C08945=1021.855,337.946,-141.506,171.172,49.202,159.657
C08946=1021.848,337.709,-141.471,171.166,49.204,159.656
C08947=1021.841,337.470,-141.437,171.159,49.205,159.655
C08948=1021.835,337.231,-141.402,171.152,49.207,159.655
C08949=1021.827,336.993,-141.367,171.146,49.209,159.654
C08950=1021.820,336.754,-141.333,171.140,49.210,159.654
C08951=1021.813,336.516,-141.298,171.134,49.211,159.653
C08952=1021.806,336.277,-141.264,171.128,49.213,159.652
C08953=1021.799,336.030,-141.228,171.121,49.214,159.652
C08954=1021.791,335.783,-141.192,171.115,49.216,159.651
C08955=1021.784,335.536,-141.157,171.108,49.218,159.651
C08956=1021.777,335.288,-141.121,171.101,49.219,159.650
C08957=1021.770,335.041,-141.086,171.095,49.221,159.649
C08958=1021.762,334.793,-141.049,171.089,49.223,159.649
C08959=1021.755,334.546,-141.014,171.082,49.225,159.648
C08960=1021.748,334.299,-140.978,171.076,49.226,159.647
C08961=1021.741,334.051,-140.943,171.070,49.228,159.647
C08962=1021.734,333.804,-140.907,171.063,49.229,159.646
C08963=1021.727,333.556,-140.871,171.057,49.231,159.646
C08964=1021.719,333.310,-140.836,171.050,49.233,159.645
C08965=1021.713,333.062,-140.800,171.044,49.235,159.645
C08966=1021.705,332.814,-140.765,171.038,49.237,159.644
C08967=1021.699,332.567,-140.730,171.031,49.238,159.643
C08968=1021.691,332.320,-140.694,171.024,49.240,159.643
C08969=1021.683,332.072,-140.659,171.018,49.242,159.642
C08970=1021.677,331.825,-140.624,171.012,49.244,159.642
C08971=1021.670,331.578,-140.589,171.006,49.246,159.641
C08972=1021.662,331.330,-140.553,171.000,49.248,159.641
C08973=1021.655,331.082,-140.519,170.993,49.250,159.640
C08974=1021.648,330.836,-140.483,170.987,49.252,159.640
C08975=1021.641,330.588,-140.448,170.980,49.253,159.639
C08976=1021.634,330.340,-140.412,170.974,49.255,159.639
C08977=1021.626,330.093,-140.378,170.968,49.257,159.638
C08978=1021.619,329.846,-140.343,170.961,49.259,159.638
C08979=1021.613,329.599,-140.307,170.955,49.261,159.637
C08980=1021.605,329.350,-140.272,170.949,49.263,159.637
C08981=1021.598,329.103,-140.237,170.943,49.265,159.636
C08982=1021.591,328.856,-140.202,170.937,49.267,159.636
C08983=1021.584,328.609,-140.167,170.930,49.269,159.635
C08984=1021.578,328.361,-140.132,170.924,49.271,159.635
C08985=1021.570,328.113,-140.098,170.918,49.272,159.634
C08986=1021.563,327.866,-140.063,170.912,49.274,159.634
C08987=1021.556,327.618,-140.028,170.906,49.276,159.633
C08988=1021.549,327.371,-139.992,170.900,49.278,159.633
C08989=1021.542,327.124,-139.958,170.894,49.280,159.632
C08990=1021.535,326.876,-139.923,170.887,49.283,159.632
C08991=1021.529,326.628,-139.888,170.881,49.285,159.631
C08992=1021.521,326.381,-139.854,170.875,49.287,159.631
C08993=1021.514,326.134,-139.819,170.869,49.289,159.630
C08994=1021.506,325.886,-139.785,170.863,49.291,159.630
C08995=1021.499,325.639,-139.750,170.856,49.294,159.630
C08996=1021.492,325.391,-139.716,170.850,49.296,159.629
C08997=1021.484,325.144,-139.682,170.844,49.298,159.629
C08998=1021.478,324.896,-139.647,170.838,49.300,159.628
C08999=1021.470,324.649,-139.613,170.832,49.302,159.628
C09000=1021.463,324.401,-139.579,170.826,49.304,159.627
C09001=1021.457,324.153,-139.544,170.819,49.306,159.627
C09002=1021.449,323.906,-139.510,170.814,49.309,159.626
C09003=1021.442,323.658,-139.476,170.808,49.311,159.626
C09004=1021.435,323.411,-139.441,170.802,49.314,159.626
C09005=1021.428,323.170,-139.408,170.796,49.315,159.625
C09006=1021.421,322.930,-139.375,170.790,49.317,159.625
C09007=1021.414,322.689,-139.342,170.784,49.320,159.624
C09008=1021.408,322.449,-139.309,170.778,49.322,159.624
C09009=1021.401,322.208,-139.275,170.773,49.325,159.624
C09010=1021.394,321.967,-139.242,170.767,49.326,159.623
C09011=1021.387,321.727,-139.209,170.761,49.329,159.623
C09012=1021.380,321.486,-139.175,170.755,49.331,159.622
C09013=1021.373,321.239,-139.142,170.749,49.334,159.622
C09014=1021.366,320.991,-139.108,170.743,49.336,159.622
C09015=1021.360,320.743,-139.073,170.737,49.338,159.621
C09016=1021.352,320.496,-139.039,170.731,49.340,159.621
C09017=1021.345,320.248,-139.005,170.726,49.343,159.621
C09018=1021.338,320.000,-138.971,170.720,49.345,159.620
C09019=1021.331,319.753,-138.937,170.713,49.347,159.620
C09020=1021.325,319.506,-138.903,170.707,49.350,159.620
C09021=1021.317,319.258,-138.870,170.701,49.352,159.619
C09022=1021.311,319.010,-138.835,170.696,49.355,159.619
C09023=1021.304,318.762,-138.801,170.690,49.357,159.619
C09024=1021.297,318.515,-138.768,170.684,49.359,159.618
C09025=1021.291,318.267,-138.733,170.678,49.362,159.618
C09026=1021.284,318.020,-138.700,170.673,49.364,159.617
C09027=1021.276,317.772,-138.666,170.667,49.367,159.617
C09028=1021.270,317.525,-138.632,170.661,49.369,159.617
C09029=1021.263,317.277,-138.598,170.655,49.371,159.616
C09030=1021.256,317.029,-138.564,170.650,49.374,159.616
C09031=1021.249,316.782,-138.530,170.644,49.377,159.616
C09032=1021.242,316.535,-138.497,170.638,49.379,159.615
C09033=1021.236,316.287,-138.462,170.632,49.381,159.615
C09034=1021.229,316.039,-138.429,170.627,49.384,159.615
C09035=1021.222,315.792,-138.396,170.620,49.387,159.614
C09036=1021.215,315.544,-138.362,170.614,49.389,159.614
C09037=1021.209,315.297,-138.328,170.609,49.392,159.614
C09038=1021.202,315.049,-138.294,170.603,49.394,159.614
C09039=1021.195,314.801,-138.260,170.597,49.396,159.613
C09040=1021.189,314.553,-138.227,170.591,49.399,159.613
C09041=1021.182,314.306,-138.193,170.585,49.401,159.613
C09042=1021.175,314.059,-138.160,170.580,49.404,159.612
C09043=1021.168,313.811,-138.126,170.574,49.407,159.612
C09044=1021.163,313.563,-138.093,170.568,49.409,159.612
C09045=1021.156,313.315,-138.059,170.563,49.412,159.611
C09046=1021.149,313.069,-138.025,170.557,49.414,159.611
C09047=1021.142,312.820,-137.992,170.551,49.417,159.611
C09048=1021.136,312.573,-137.958,170.546,49.420,159.611
C09049=1021.129,312.325,-137.924,170.540,49.422,159.610
C09050=1021.123,312.078,-137.892,170.534,49.425,159.610
C09051=1021.115,311.830,-137.858,170.529,49.427,159.610
C09052=1021.109,311.582,-137.825,170.523,49.430,159.609
C09053=1021.103,311.334,-137.791,170.517,49.433,159.609
C09054=1021.096,311.087,-137.758,170.512,49.435,159.609
C09055=1021.090,310.840,-137.724,170.506,49.438,159.609
C09056=1021.083,310.592,-137.691,170.502,49.441,159.608
C09057=1021.077,310.344,-137.657,170.496,49.443,159.608
C09058=1021.070,310.096,-137.624,170.490,49.446,159.608
C09059=1021.064,309.849,-137.591,170.485,49.448,159.608
C09060=1021.057,309.602,-137.558,170.478,49.452,159.607
C09061=1021.050,309.353,-137.525,170.473,49.455,159.607
C09062=1021.043,309.106,-137.493,170.467,49.458,159.607
C09063=1021.036,308.858,-137.460,170.462,49.460,159.607
C09064=1021.029,308.610,-137.427,170.456,49.463,159.606
C09065=1021.023,308.372,-137.396,170.451,49.466,159.606
C09066=1021.016,308.134,-137.364,170.446,49.468,159.606
C09067=1021.009,307.896,-137.333,170.441,49.472,159.606
C09068=1021.003,307.658,-137.301,170.435,49.474,159.606
C09069=1020.996,307.420,-137.270,170.429,49.477,159.606
C09070=1020.990,307.182,-137.238,170.424,49.480,159.605
C09071=1020.984,306.944,-137.207,170.419,49.482,159.605
C09072=1020.977,306.706,-137.176,170.414,49.486,159.605
C09073=1020.970,306.459,-137.144,170.409,49.488,159.605
C09074=1020.963,306.210,-137.111,170.403,49.491,159.605
C09075=1020.956,305.963,-137.079,170.398,49.495,159.605
C09076=1020.950,305.715,-137.046,170.392,49.497,159.604
C09077=1020.943,305.467,-137.013,170.387,49.501,159.604
C09078=1020.936,305.220,-136.981,170.381,49.503,159.604
C09079=1020.930,304.972,-136.948,170.376,49.506,159.604
C09080=1020.922,304.724,-136.916,170.371,49.510,159.604
C09081=1020.916,304.476,-136.883,170.365,49.512,159.603
C09082=1020.910,304.229,-136.851,170.360,49.515,159.603
C09083=1020.903,303.981,-136.818,170.354,49.519,159.603
C09084=1020.896,303.734,-136.786,170.349,49.521,159.603
C09085=1020.889,303.485,-136.754,170.343,49.525,159.603
C09086=1020.883,303.237,-136.721,170.338,49.528,159.603
C09087=1020.876,302.990,-136.688,170.333,49.531,159.603
C09088=1020.869,302.743,-136.656,170.327,49.534,159.602
C09089=1020.863,302.494,-136.624,170.322,49.537,159.602
C09090=1020.856,302.246,-136.592,170.316,49.540,159.602
C09091=1020.849,301.999,-136.559,170.311,49.543,159.602
C09092=1020.843,301.751,-136.527,170.306,49.547,159.602
C09093=1020.836,301.503,-136.495,170.300,49.549,159.602
C09094=1020.830,301.256,-136.462,170.295,49.552,159.602
C09095=1020.823,301.008,-136.431,170.290,49.556,159.602
C09096=1020.817,300.760,-136.398,170.284,49.559,159.601
C09097=1020.810,300.512,-136.365,170.279,49.562,159.601
C09098=1020.803,300.264,-136.333,170.274,49.565,159.601
C09099=1020.797,300.016,-136.301,170.268,49.568,159.601
C09100=1020.790,299.768,-136.269,170.263,49.571,159.601
C09101=1020.784,299.521,-136.236,170.257,49.575,159.601
C09102=1020.778,299.273,-136.204,170.252,49.578,159.601
C09103=1020.771,299.025,-136.172,170.247,49.581,159.601
C09104=1020.765,298.777,-136.140,170.241,49.584,159.600
C09105=1020.758,298.530,-136.108,170.236,49.588,159.600
C09106=1020.752,298.282,-136.076,170.231,49.591,159.600
C09107=1020.745,298.034,-136.044,170.225,49.594,159.600
C09108=1020.739,297.786,-136.012,170.220,49.597,159.600
C09109=1020.733,297.538,-135.980,170.215,49.601,159.600
C09110=1020.726,297.291,-135.948,170.211,49.603,159.600
C09111=1020.720,297.042,-135.916,170.205,49.607,159.600
C09112=1020.713,296.795,-135.884,170.200,49.610,159.600
C09113=1020.707,296.547,-135.851,170.195,49.613,159.600
C09114=1020.700,296.299,-135.820,170.189,49.617,159.600
C09115=1020.694,296.051,-135.788,170.184,49.620,159.599
C09116=1020.689,295.804,-135.756,170.179,49.623,159.599
C09117=1020.682,295.556,-135.724,170.174,49.627,159.599
C09118=1020.676,295.308,-135.692,170.168,49.630,159.599
C09119=1020.669,295.061,-135.660,170.163,49.633,159.599
C09120=1020.663,294.812,-135.628,170.158,49.637,159.599
C09121=1020.657,294.564,-135.596,170.153,49.640,159.599
C09122=1020.650,294.316,-135.565,170.148,49.643,159.599
C09123=1020.644,294.068,-135.533,170.143,49.647,159.599
C09124=1020.638,293.821,-135.501,170.138,49.650,159.599
C09125=1020.632,293.592,-135.471,170.133,49.653,159.599
C09126=1020.627,293.362,-135.442,170.128,49.656,159.599
C09127=1020.620,293.133,-135.413,170.123,49.659,159.599
C09128=1020.614,292.904,-135.384,170.119,49.662,159.599
C09129=1020.608,292.674,-135.355,170.113,49.666,159.599
C09130=1020.603,292.445,-135.325,170.110,49.669,159.599
C09131=1020.596,292.216,-135.296,170.104,49.673,159.599
C09132=1020.590,291.986,-135.268,170.100,49.675,159.599
C09133=1020.584,291.738,-135.236,170.095,49.679,159.599
C09134=1020.578,291.490,-135.204,170.090,49.683,159.599
C09135=1020.571,291.242,-135.173,170.084,49.686,159.599
C09136=1020.565,290.995,-135.142,170.079,49.690,159.599
C09137=1020.558,290.747,-135.110,170.074,49.693,159.599
C09138=1020.552,290.499,-135.079,170.069,49.697,159.599
C09139=1020.545,290.251,-135.048,170.064,49.700,159.599
C09140=1020.539,290.004,-135.017,170.059,49.704,159.599
C09141=1020.533,289.756,-134.985,170.054,49.707,159.599
C09142=1020.526,289.507,-134.954,170.049,49.711,159.599
C09143=1020.520,289.259,-134.923,170.044,49.715,159.599
C09144=1020.514,289.012,-134.892,170.038,49.719,159.599
C09145=1020.507,288.763,-134.861,170.034,49.722,159.599
C09146=1020.500,288.515,-134.830,170.028,49.726,159.599
C09147=1020.494,288.268,-134.798,170.023,49.730,159.599
C09148=1020.488,288.020,-134.768,170.018,49.734,159.599
C09149=1020.481,287.772,-134.736,170.014,49.736,159.599
C09150=1020.474,287.524,-134.705,170.009,49.740,159.599
C09151=1020.469,287.276,-134.675,170.004,49.744,159.599
C09152=1020.462,287.028,-134.643,169.999,49.748,159.599
C09153=1020.455,286.780,-134.612,169.994,49.752,159.599
C09154=1020.449,286.533,-134.581,169.989,49.755,159.599
C09155=1020.443,286.284,-134.551,169.984,49.759,159.599
C09156=1020.436,286.036,-134.519,169.979,49.763,159.599
C09157=1020.430,285.788,-134.489,169.974,49.767,159.599
C09158=1020.424,285.540,-134.457,169.969,49.771,159.599
C09159=1020.417,285.292,-134.427,169.964,49.774,159.599
C09160=1020.411,285.045,-134.396,169.959,49.778,159.599
C09161=1020.405,284.796,-134.365,169.954,49.782,159.600
C09162=1020.399,284.548,-134.335,169.949,49.786,159.599
C09163=1020.392,284.300,-134.303,169.944,49.789,159.600
C09164=1020.386,284.052,-134.272,169.939,49.793,159.600
C09165=1020.379,283.804,-134.243,169.934,49.797,159.600
C09166=1020.373,283.556,-134.212,169.929,49.801,159.600
C09167=1020.367,283.309,-134.181,169.924,49.805,159.600
C09168=1020.360,283.060,-134.150,169.919,49.809,159.600
C09169=1020.354,282.812,-134.119,169.914,49.813,159.600
C09170=1020.347,282.564,-134.090,169.909,49.817,159.600
C09171=1020.341,282.316,-134.058,169.904,49.821,159.600
C09172=1020.335,282.068,-134.028,169.899,49.825,159.600
C09173=1020.328,281.820,-133.997,169.895,49.829,159.600
C09174=1020.322,281.572,-133.967,169.890,49.833,159.600
C09175=1020.315,281.324,-133.937,169.886,49.836,159.601
C09176=1020.309,281.076,-133.906,169.881,49.840,159.601
C09177=1020.303,280.827,-133.876,169.876,49.845,159.601
C09178=1020.297,280.580,-133.845,169.871,49.849,159.601
C09179=1020.290,280.332,-133.814,169.866,49.853,159.601
C09180=1020.284,280.084,-133.784,169.861,49.857,159.601
C09181=1020.278,279.836,-133.753,169.856,49.861,159.601
C09182=1020.272,279.588,-133.723,169.852,49.865,159.601
C09183=1020.265,279.340,-133.693,169.847,49.868,159.602
C09184=1020.259,279.092,-133.663,169.842,49.872,159.602
C09185=1020.254,278.869,-133.635,169.838,49.876,159.602
C09186=1020.247,278.645,-133.608,169.833,49.880,159.602
C09187=1020.242,278.422,-133.581,169.829,49.884,159.602
C09188=1020.237,278.199,-133.553,169.825,49.887,159.602
C09189=1020.231,277.976,-133.526,169.820,49.891,159.602
C09190=1020.226,277.753,-133.499,169.816,49.895,159.603
C09191=1020.219,277.529,-133.472,169.812,49.898,159.603
C09192=1020.214,277.306,-133.444,169.807,49.902,159.603
C09193=1020.209,277.058,-133.414,169.802,49.906,159.603
C09194=1020.201,276.810,-133.384,169.797,49.910,159.603
C09195=1020.196,276.562,-133.353,169.792,49.914,159.603
C09196=1020.189,276.314,-133.324,169.788,49.919,159.603
C09197=1020.183,276.066,-133.293,169.783,49.923,159.603
C09198=1020.176,275.818,-133.264,169.778,49.927,159.604
C09199=1020.171,275.570,-133.234,169.774,49.931,159.604
C09200=1020.163,275.322,-133.203,169.769,49.935,159.604
C09201=1020.158,275.073,-133.174,169.764,49.940,159.604
C09202=1020.152,274.825,-133.143,169.759,49.944,159.604
C09203=1020.145,274.577,-133.113,169.755,49.948,159.604
C09204=1020.139,274.329,-133.084,169.751,49.952,159.605
C09205=1020.133,274.081,-133.054,169.746,49.957,159.605
C09206=1020.126,273.833,-133.023,169.741,49.961,159.605
C09207=1020.120,273.584,-132.994,169.737,49.965,159.605
C09208=1020.114,273.337,-132.964,169.732,49.969,159.605
C09209=1020.107,273.088,-132.934,169.727,49.974,159.606
C09210=1020.102,272.840,-132.904,169.722,49.978,159.606
C09211=1020.095,272.592,-132.874,169.718,49.982,159.606
C09212=1020.090,272.344,-132.845,169.713,49.986,159.606
C09213=1020.082,272.096,-132.815,169.708,49.991,159.606
C09214=1020.076,271.848,-132.786,169.704,49.995,159.607
C09215=1020.070,271.600,-132.755,169.699,49.999,159.607
C09216=1020.064,271.352,-132.726,169.694,50.004,159.607
C09217=1020.058,271.103,-132.696,169.690,50.009,159.607
C09218=1020.051,270.855,-132.666,169.685,50.013,159.607
C09219=1020.046,270.607,-132.637,169.680,50.017,159.608
C09220=1020.039,270.359,-132.607,169.676,50.022,159.608
C09221=1020.033,270.111,-132.578,169.671,50.026,159.608
C09222=1020.027,269.862,-132.547,169.666,50.030,159.608
C09223=1020.020,269.614,-132.518,169.662,50.035,159.609
C09224=1020.015,269.366,-132.489,169.657,50.039,159.609
C09225=1020.009,269.118,-132.460,169.652,50.044,159.609
C09226=1020.002,268.870,-132.430,169.648,50.048,159.609
C09227=1019.996,268.622,-132.401,169.643,50.053,159.610
C09228=1019.990,268.373,-132.371,169.638,50.057,159.610
C09229=1019.984,268.125,-132.342,169.634,50.061,159.610
C09230=1019.977,267.877,-132.312,169.629,50.066,159.610
C09231=1019.971,267.629,-132.282,169.624,50.071,159.610
C09232=1019.965,267.381,-132.253,169.620,50.075,159.611
C09233=1019.959,267.133,-132.224,169.615,50.080,159.611
C09234=1019.953,266.885,-132.195,169.611,50.085,159.611
C09235=1019.946,266.636,-132.164,169.606,50.089,159.612
C09236=1019.940,266.388,-132.135,169.602,50.094,159.612
C09237=1019.934,266.140,-132.106,169.597,50.098,159.612
C09238=1019.928,265.892,-132.077,169.593,50.103,159.612
C09239=1019.921,265.643,-132.048,169.588,50.107,159.612
C09240=1019.916,265.395,-132.019,169.583,50.112,159.613
C09241=1019.910,265.147,-131.990,169.579,50.116,159.613
C09242=1019.903,264.899,-131.961,169.574,50.121,159.613
C09243=1019.897,264.651,-131.932,169.570,50.126,159.614
C09244=1019.891,264.402,-131.903,169.565,50.131,159.614
C09245=1019.885,264.182,-131.876,169.560,50.135,159.614
C09246=1019.880,263.961,-131.851,169.557,50.139,159.615
C09247=1019.874,263.740,-131.825,169.553,50.143,159.615
C09248=1019.868,263.519,-131.799,169.548,50.147,159.615
C09249=1019.863,263.298,-131.773,169.545,50.152,159.615
C09250=1019.857,263.078,-131.747,169.541,50.155,159.615
C09251=1019.852,262.856,-131.722,169.537,50.160,159.616
C09252=1019.846,262.636,-131.696,169.533,50.164,159.616
C09253=1019.841,262.387,-131.666,169.528,50.169,159.616
C09254=1019.835,262.139,-131.637,169.524,50.174,159.617
C09255=1019.829,261.890,-131.609,169.519,50.178,159.617
C09256=1019.822,261.642,-131.580,169.515,50.183,159.617
C09257=1019.816,261.394,-131.551,169.511,50.188,159.618
C09258=1019.810,261.146,-131.522,169.506,50.193,159.618
C09259=1019.804,260.898,-131.493,169.502,50.198,159.618
C09260=1019.798,260.649,-131.464,169.497,50.202,159.619
C09261=1019.791,260.401,-131.435,169.493,50.207,159.619
C09262=1019.785,260.153,-131.406,169.488,50.212,159.619
C09263=1019.779,259.905,-131.377,169.484,50.217,159.620
C09264=1019.773,259.656,-131.349,169.478,50.222,159.620
C09265=1019.766,259.408,-131.320,169.474,50.227,159.620
C09266=1019.760,259.159,-131.292,169.470,50.232,159.620
C09267=1019.754,258.912,-131.263,169.465,50.237,159.621
C09268=1019.748,258.664,-131.236,169.461,50.242,159.621
C09269=1019.741,258.415,-131.207,169.457,50.247,159.622
C09270=1019.736,258.167,-131.178,169.452,50.252,159.622
C09271=1019.729,257.919,-131.150,169.448,50.257,159.622
C09272=1019.723,257.670,-131.121,169.444,50.262,159.623
C09273=1019.716,257.422,-131.092,169.438,50.267,159.623
C09274=1019.710,257.173,-131.065,169.434,50.272,159.623
C09275=1019.703,256.925,-131.036,169.430,50.277,159.624
C09276=1019.697,256.677,-131.007,169.425,50.282,159.624
C09277=1019.690,256.429,-130.979,169.421,50.287,159.625
C09278=1019.685,256.180,-130.951,169.417,50.293,159.625
C09279=1019.679,255.932,-130.923,169.412,50.297,159.625
C09280=1019.672,255.684,-130.894,169.408,50.303,159.626
C09281=1019.666,255.435,-130.866,169.403,50.308,159.626
C09282=1019.660,255.187,-130.838,169.399,50.313,159.627
C09283=1019.653,254.939,-130.809,169.394,50.318,159.627
C09284=1019.647,254.690,-130.781,169.390,50.323,159.627
C09285=1019.642,254.442,-130.753,169.386,50.328,159.628
C09286=1019.635,254.194,-130.724,169.381,50.333,159.628
C09287=1019.629,253.945,-130.696,169.377,50.338,159.628
C09288=1019.623,253.697,-130.668,169.373,50.343,159.629
C09289=1019.616,253.448,-130.640,169.368,50.348,159.629
C09290=1019.611,253.201,-130.611,169.363,50.354,159.630
C09291=1019.605,252.952,-130.583,169.359,50.359,159.630
C09292=1019.598,252.704,-130.555,169.355,50.364,159.631
C09293=1019.592,252.455,-130.527,169.350,50.369,159.631
C09294=1019.586,252.207,-130.498,169.346,50.374,159.631
C09295=1019.580,251.959,-130.470,169.342,50.380,159.632
C09296=1019.574,251.710,-130.442,169.338,50.385,159.632
C09297=1019.568,251.461,-130.414,169.333,50.390,159.633
C09298=1019.562,251.214,-130.386,169.329,50.395,159.633
C09299=1019.556,250.966,-130.357,169.324,50.401,159.633
C09300=1019.550,250.717,-130.329,169.320,50.406,159.634
C09301=1019.543,250.468,-130.301,169.316,50.411,159.634
C09302=1019.538,250.220,-130.273,169.311,50.416,159.635
C09303=1019.532,249.972,-130.245,169.307,50.422,159.635
C09304=1019.525,249.723,-130.217,169.303,50.427,159.636
C09305=1019.520,249.502,-130.192,169.299,50.432,159.636
C09306=1019.515,249.280,-130.167,169.295,50.437,159.636
C09307=1019.510,249.058,-130.143,169.292,50.441,159.637
C09308=1019.504,248.837,-130.117,169.287,50.446,159.637
C09309=1019.499,248.614,-130.092,169.284,50.451,159.638
C09310=1019.493,248.393,-130.067,169.280,50.455,159.638
C09311=1019.488,248.171,-130.042,169.276,50.460,159.638
C09312=1019.483,247.950,-130.017,169.272,50.465,159.639
C09313=1019.476,247.702,-129.989,169.268,50.470,159.639
C09314=1019.471,247.454,-129.961,169.264,50.476,159.640
C09315=1019.464,247.205,-129.933,169.260,50.481,159.640
C09316=1019.458,246.956,-129.906,169.256,50.486,159.641
C09317=1019.453,246.708,-129.878,169.251,50.491,159.641
C09318=1019.446,246.459,-129.850,169.247,50.496,159.641
C09319=1019.441,246.211,-129.822,169.242,50.502,159.642
C09320=1019.435,245.962,-129.794,169.238,50.508,159.642
C09321=1019.429,245.714,-129.766,169.234,50.513,159.643
C09322=1019.423,245.466,-129.738,169.229,50.518,159.643
C09323=1019.417,245.217,-129.710,169.225,50.524,159.643
C09324=1019.411,244.969,-129.682,169.221,50.529,159.644
C09325=1019.405,244.721,-129.654,169.217,50.534,159.644
C09326=1019.399,244.473,-129.627,169.213,50.540,159.645
C09327=1019.393,244.224,-129.599,169.209,50.546,159.646
C09328=1019.388,243.976,-129.571,169.204,50.551,159.646
C09329=1019.381,243.727,-129.543,169.200,50.557,159.646
C09330=1019.376,243.479,-129.515,169.196,50.562,159.647
C09331=1019.370,243.230,-129.487,169.192,50.567,159.647
C09332=1019.364,242.982,-129.460,169.188,50.573,159.648
C09333=1019.358,242.733,-129.433,169.184,50.578,159.648
C09334=1019.352,242.485,-129.405,169.180,50.584,159.649
C09335=1019.346,242.236,-129.378,169.175,50.590,159.649
C09336=1019.340,241.989,-129.350,169.171,50.595,159.650
C09337=1019.334,241.740,-129.322,169.166,50.601,159.650
C09338=1019.328,241.492,-129.295,169.163,50.607,159.651
C09339=1019.322,241.243,-129.268,169.159,50.612,159.651
C09340=1019.316,240.994,-129.240,169.153,50.618,159.652
C09341=1019.310,240.746,-129.213,169.150,50.624,159.652
C09342=1019.304,240.498,-129.185,169.146,50.629,159.653
C09343=1019.298,240.249,-129.158,169.141,50.635,159.653
C09344=1019.292,240.001,-129.130,169.138,50.641,159.654
C09345=1019.286,239.753,-129.104,169.133,50.646,159.654
C09346=1019.280,239.504,-129.075,169.129,50.652,159.655
C09347=1019.275,239.256,-129.049,169.125,50.658,159.656
C09348=1019.268,239.007,-129.021,169.121,50.663,159.656
C09349=1019.262,238.759,-128.994,169.117,50.669,159.657
C09350=1019.256,238.510,-128.966,169.112,50.675,159.657
C09351=1019.250,238.262,-128.939,169.108,50.681,159.658
C09352=1019.245,238.013,-128.913,169.104,50.686,159.658
C09353=1019.238,237.765,-128.885,169.100,50.692,159.659
C09354=1019.232,237.517,-128.858,169.095,50.698,159.659
C09355=1019.226,237.268,-128.831,169.091,50.704,159.660
C09356=1019.220,237.020,-128.804,169.087,50.710,159.660
C09357=1019.214,236.771,-128.777,169.083,50.716,159.661
C09358=1019.208,236.522,-128.750,169.079,50.722,159.662
C09359=1019.202,236.274,-128.724,169.075,50.727,159.662
C09360=1019.195,236.026,-128.696,169.071,50.734,159.663
C09361=1019.189,235.777,-128.669,169.066,50.739,159.663
C09362=1019.184,235.529,-128.643,169.062,50.745,159.664
C09363=1019.177,235.280,-128.616,169.059,50.751,159.664
C09364=1019.171,235.032,-128.588,169.054,50.757,159.665
C09365=1019.166,234.807,-128.564,169.051,50.763,159.666
C09366=1019.160,234.581,-128.540,169.047,50.768,159.666
C09367=1019.155,234.356,-128.515,169.043,50.774,159.667
C09368=1019.150,234.132,-128.491,169.039,50.779,159.667
C09369=1019.145,233.907,-128.467,169.035,50.784,159.668
C09370=1019.139,233.682,-128.442,169.031,50.790,159.668
C09371=1019.134,233.457,-128.418,169.029,50.795,159.669
C09372=1019.128,233.232,-128.394,169.024,50.801,159.669
C09373=1019.122,232.983,-128.367,169.021,50.807,159.670
C09374=1019.116,232.735,-128.340,169.016,50.812,159.670
C09375=1019.110,232.487,-128.314,169.012,50.819,159.671
C09376=1019.104,232.238,-128.287,169.008,50.825,159.672
C09377=1019.098,231.989,-128.260,169.004,50.831,159.672
C09378=1019.092,231.741,-128.233,169.000,50.837,159.673
C09379=1019.086,231.493,-128.206,168.996,50.843,159.673
C09380=1019.080,231.245,-128.179,168.992,50.849,159.674
C09381=1019.074,230.996,-128.152,168.987,50.855,159.675
C09382=1019.068,230.747,-128.126,168.984,50.861,159.675
C09383=1019.062,230.499,-128.099,168.980,50.867,159.676
C09384=1019.057,230.251,-128.072,168.975,50.874,159.676
C09385=1019.050,230.001,-128.045,168.972,50.880,159.677
C09386=1019.044,229.753,-128.019,168.968,50.886,159.678
C09387=1019.039,229.504,-127.993,168.963,50.892,159.678
C09388=1019.033,229.256,-127.966,168.959,50.898,159.679
C09389=1019.027,229.007,-127.939,168.955,50.904,159.680
C09390=1019.020,228.759,-127.913,168.951,50.910,159.680
C09391=1019.015,228.510,-127.886,168.947,50.916,159.681
C09392=1019.009,228.262,-127.860,168.943,50.922,159.681
C09393=1019.003,228.014,-127.833,168.939,50.929,159.682
C09394=1018.997,227.765,-127.806,168.935,50.935,159.683
C09395=1018.992,227.516,-127.780,168.932,50.942,159.684
C09396=1018.985,227.268,-127.754,168.927,50.948,159.684
C09397=1018.979,227.019,-127.727,168.923,50.954,159.685
C09398=1018.973,226.771,-127.701,168.919,50.961,159.685
C09399=1018.968,226.522,-127.675,168.915,50.967,159.686
C09400=1018.961,226.274,-127.649,168.911,50.973,159.687
C09401=1018.955,226.025,-127.622,168.906,50.979,159.687
C09402=1018.950,225.777,-127.595,168.903,50.985,159.688
C09403=1018.943,225.528,-127.570,168.899,50.993,159.689
C09404=1018.937,225.279,-127.543,168.895,50.999,159.689
C09405=1018.931,225.031,-127.518,168.890,51.005,159.690
C09406=1018.925,224.782,-127.491,168.886,51.011,159.691
C09407=1018.919,224.534,-127.464,168.883,51.018,159.692
C09408=1018.913,224.285,-127.439,168.879,51.024,159.692
C09409=1018.907,224.037,-127.412,168.875,51.031,159.693
C09410=1018.901,223.788,-127.387,168.871,51.038,159.694
C09411=1018.895,223.539,-127.360,168.867,51.044,159.694
C09412=1018.889,223.290,-127.334,168.862,51.050,159.695
C09413=1018.883,223.042,-127.308,168.859,51.056,159.695
C09414=1018.877,222.793,-127.282,168.855,51.063,159.696
C09415=1018.871,222.545,-127.256,168.851,51.070,159.697
C09416=1018.865,222.296,-127.230,168.847,51.076,159.698
C09417=1018.859,222.048,-127.204,168.843,51.083,159.698
C09418=1018.853,221.799,-127.178,168.839,51.089,159.699
C09419=1018.847,221.551,-127.152,168.835,51.096,159.700
C09420=1018.841,221.302,-127.126,168.831,51.102,159.700
C09421=1018.835,221.054,-127.100,168.826,51.109,159.701
C09422=1018.830,220.805,-127.074,168.823,51.116,159.702
C09423=1018.824,220.557,-127.048,168.818,51.122,159.702
C09424=1018.818,220.308,-127.022,168.815,51.129,159.703
C09425=1018.812,220.079,-126.998,168.811,51.135,159.704
C09426=1018.807,219.850,-126.974,168.808,51.141,159.705
C09427=1018.801,219.621,-126.950,168.804,51.147,159.705
C09428=1018.796,219.392,-126.926,168.801,51.153,159.706
C09429=1018.790,219.163,-126.902,168.796,51.159,159.706
C09430=1018.785,218.933,-126.878,168.793,51.165,159.707
C09431=1018.779,218.704,-126.854,168.789,51.171,159.708
C09432=1018.774,218.475,-126.830,168.785,51.177,159.708
C09433=1018.768,218.226,-126.804,168.782,51.184,159.709
C09434=1018.762,217.978,-126.779,168.778,51.191,159.710
C09435=1018.757,217.730,-126.754,168.774,51.197,159.711
C09436=1018.750,217.482,-126.728,168.770,51.204,159.712
C09437=1018.745,217.233,-126.702,168.767,51.211,159.712
C09438=1018.738,216.984,-126.676,168.762,51.218,159.713
C09439=1018.732,216.735,-126.651,168.758,51.225,159.714
C09440=1018.727,216.486,-126.625,168.755,51.232,159.715
C09441=1018.720,216.238,-126.599,168.750,51.238,159.715
C09442=1018.714,215.990,-126.574,168.747,51.245,159.716
C09443=1018.708,215.741,-126.548,168.742,51.252,159.717
C09444=1018.702,215.492,-126.522,168.739,51.259,159.718
C09445=1018.696,215.243,-126.497,168.735,51.265,159.718
C09446=1018.690,214.995,-126.472,168.730,51.273,159.719
C09447=1018.684,214.746,-126.446,168.727,51.279,159.720
C09448=1018.678,214.497,-126.420,168.723,51.287,159.721
C09449=1018.673,214.249,-126.395,168.720,51.293,159.722
C09450=1018.666,214.000,-126.370,168.715,51.300,159.722
C09451=1018.661,213.752,-126.343,168.712,51.307,159.723
C09452=1018.654,213.503,-126.318,168.707,51.314,159.724
C09453=1018.648,213.255,-126.293,168.703,51.321,159.725
C09454=1018.643,213.006,-126.267,168.700,51.328,159.725
C09455=1018.637,212.757,-126.241,168.696,51.335,159.726
C09456=1018.630,212.508,-126.216,168.692,51.341,159.727
C09457=1018.625,212.260,-126.191,168.688,51.349,159.728
C09458=1018.619,212.011,-126.165,168.684,51.356,159.728
C09459=1018.613,211.763,-126.140,168.680,51.363,159.729
C09460=1018.607,211.514,-126.115,168.676,51.370,159.730
C09461=1018.601,211.265,-126.089,168.673,51.377,159.731
C09462=1018.596,211.017,-126.064,168.669,51.384,159.732
C09463=1018.590,210.768,-126.038,168.664,51.391,159.733
C09464=1018.584,210.519,-126.014,168.661,51.398,159.733
C09465=1018.578,210.270,-125.988,168.657,51.405,159.734
C09466=1018.572,210.021,-125.962,168.654,51.412,159.735
C09467=1018.566,209.774,-125.937,168.650,51.419,159.736
C09468=1018.560,209.525,-125.912,168.645,51.426,159.737
C09469=1018.554,209.276,-125.887,168.642,51.433,159.738
C09470=1018.548,209.028,-125.861,168.638,51.440,159.738
C09471=1018.542,208.778,-125.837,168.634,51.448,159.739
C09472=1018.537,208.530,-125.811,168.631,51.454,159.740
C09473=1018.531,208.281,-125.786,168.626,51.462,159.741
C09474=1018.525,208.033,-125.761,168.622,51.469,159.741
C09475=1018.518,207.784,-125.735,168.618,51.477,159.742
C09476=1018.513,207.535,-125.711,168.615,51.484,159.743
C09477=1018.507,207.287,-125.686,168.611,51.491,159.744
C09478=1018.501,207.038,-125.660,168.607,51.498,159.745
C09479=1018.495,206.789,-125.636,168.603,51.505,159.746
C09480=1018.489,206.541,-125.611,168.600,51.513,159.747
C09481=1018.483,206.292,-125.585,168.595,51.520,159.748
C09482=1018.477,206.043,-125.561,168.591,51.527,159.748
C09483=1018.472,205.795,-125.536,168.588,51.534,159.749
C09484=1018.465,205.546,-125.510,168.584,51.542,159.750
C09485=1018.460,205.317,-125.488,168.581,51.548,159.751
C09486=1018.454,205.087,-125.465,168.577,51.555,159.752
C09487=1018.449,204.858,-125.441,168.573,51.562,159.752
C09488=1018.444,204.629,-125.419,168.570,51.569,159.753
C09489=1018.438,204.400,-125.397,168.566,51.575,159.754
C09490=1018.432,204.171,-125.374,168.563,51.582,159.755
C09491=1018.426,203.942,-125.350,168.559,51.589,159.756
C09492=1018.400,202.697,-125.232,168.087,51.498,159.649
C09493=1018.396,202.448,-125.209,168.082,51.506,159.650
C09494=1018.390,202.199,-125.186,168.078,51.514,159.651
C09495=1018.385,201.950,-125.163,168.073,51.523,159.652
C09496=1018.381,201.701,-125.140,168.069,51.532,159.653
C09497=1018.376,201.452,-125.117,168.064,51.540,159.653
C09498=1018.371,201.204,-125.094,168.060,51.548,159.654
C09499=1018.366,200.954,-125.071,168.055,51.556,159.655
C09500=1018.361,200.705,-125.047,168.051,51.565,159.656
C09501=1018.356,200.457,-125.024,168.046,51.573,159.657
C09502=1018.351,200.208,-125.001,168.041,51.582,159.658
C09503=1018.346,199.959,-124.978,168.037,51.590,159.659
C09504=1018.341,199.710,-124.955,168.033,51.599,159.660
C09505=1018.336,199.461,-124.931,168.028,51.607,159.661
C09506=1018.332,199.212,-124.909,168.023,51.616,159.662
C09507=1018.326,198.963,-124.886,168.019,51.624,159.663
C09508=1018.321,198.715,-124.863,168.014,51.632,159.663
C09509=1018.316,198.465,-124.840,168.010,51.641,159.664
C09510=1018.311,198.217,-124.818,168.005,51.649,159.665
C09511=1018.305,197.968,-124.795,168.001,51.658,159.666
C09512=1018.301,197.718,-124.772,167.997,51.666,159.667
C09513=1018.295,197.470,-124.750,167.992,51.675,159.668
C09514=1018.290,197.221,-124.727,167.988,51.684,159.669
C09515=1018.286,196.972,-124.704,167.983,51.693,159.670
C09516=1018.280,196.723,-124.681,167.978,51.701,159.671
C09517=1018.275,196.474,-124.659,167.975,51.710,159.672
C09518=1018.270,196.225,-124.636,167.970,51.718,159.673
C09519=1018.265,195.976,-124.614,167.966,51.727,159.674
C09520=1018.259,195.727,-124.591,167.961,51.735,159.675
C09521=1018.254,195.479,-124.568,167.956,51.744,159.676
C09522=1018.250,195.229,-124.546,167.953,51.752,159.677
C09523=1018.245,194.981,-124.523,167.948,51.761,159.678
C09524=1018.239,194.732,-124.501,167.943,51.770,159.678
C09525=1018.235,194.483,-124.478,167.939,51.779,159.679
C09526=1018.229,194.234,-124.455,167.935,51.787,159.680
C09527=1018.224,193.985,-124.433,167.931,51.796,159.681
C09528=1018.219,193.736,-124.410,167.926,51.804,159.682
C09529=1018.215,193.487,-124.388,167.922,51.813,159.683
C09530=1018.210,193.239,-124.365,167.918,51.821,159.684
C09531=1018.205,192.989,-124.343,167.913,51.830,159.685
C09532=1018.200,192.741,-124.320,167.908,51.838,159.686
C09533=1018.194,192.491,-124.298,167.905,51.847,159.687
C09534=1018.189,192.243,-124.275,167.900,51.856,159.688
C09535=1018.185,191.994,-124.253,167.896,51.865,159.689
C09536=1018.180,191.744,-124.231,167.892,51.873,159.690
C09537=1018.175,191.496,-124.208,167.887,51.882,159.691
C09538=1018.170,191.246,-124.185,167.883,51.890,159.692
C09539=1018.165,190.998,-124.163,167.879,51.899,159.693
C09540=1018.160,190.749,-124.141,167.874,51.907,159.694
C09541=1018.155,190.499,-124.118,167.870,51.916,159.695
C09542=1018.150,190.251,-124.095,167.866,51.924,159.696
C09543=1018.145,190.002,-124.073,167.862,51.933,159.697
C09544=1018.140,189.753,-124.051,167.857,51.941,159.698
C09545=1018.136,189.504,-124.029,167.854,51.950,159.699
C09546=1018.131,189.256,-124.006,167.849,51.959,159.699
C09547=1018.125,189.006,-123.984,167.845,51.968,159.701
C09548=1018.121,188.757,-123.962,167.841,51.976,159.702
C09549=1018.116,188.509,-123.939,167.836,51.985,159.702
C09550=1018.111,188.259,-123.917,167.832,51.994,159.704
C09551=1018.106,188.010,-123.894,167.828,52.002,159.704
C09552=1018.102,187.761,-123.872,167.824,52.011,159.705
C09553=1018.096,187.481,-123.847,167.819,52.020,159.706
C09554=1018.090,187.199,-123.822,167.814,52.030,159.708
C09555=1018.085,186.919,-123.797,167.810,52.039,159.709
C09556=1018.080,186.638,-123.772,167.805,52.049,159.710
C09557=1018.075,186.390,-123.749,167.801,52.058,159.711
C09558=1018.070,186.140,-123.727,167.797,52.066,159.712
C09559=1018.065,185.892,-123.705,167.793,52.075,159.713
C09560=1018.060,185.643,-123.683,167.789,52.083,159.714
C09561=1018.055,185.394,-123.661,167.785,52.093,159.715
C09562=1018.051,185.145,-123.639,167.781,52.101,159.716
C09563=1018.046,184.896,-123.616,167.776,52.110,159.717
C09564=1018.041,184.647,-123.594,167.772,52.118,159.717
C09565=1018.037,184.398,-123.571,167.768,52.127,159.719
C09566=1018.032,184.149,-123.549,167.764,52.135,159.719
C09567=1018.027,183.900,-123.528,167.760,52.144,159.721
C09568=1018.022,183.651,-123.505,167.755,52.152,159.721
C09569=1018.018,183.402,-123.483,167.752,52.161,159.723
C09570=1018.013,183.153,-123.461,167.747,52.170,159.723
C09571=1018.008,182.904,-123.439,167.744,52.178,159.724
C09572=1018.003,182.655,-123.417,167.739,52.187,159.725
C09573=1017.999,182.406,-123.395,167.736,52.195,159.726
C09574=1017.994,182.157,-123.373,167.731,52.204,159.727
C09575=1017.989,181.908,-123.351,167.728,52.213,159.728
C09576=1017.984,181.659,-123.329,167.723,52.222,159.729
C09577=1017.979,181.410,-123.307,167.719,52.231,159.730
C09578=1017.974,181.161,-123.286,167.715,52.239,159.731
C09579=1017.968,180.912,-123.264,167.711,52.248,159.732
C09580=1017.964,180.663,-123.242,167.707,52.257,159.733
C09581=1017.958,180.414,-123.222,167.703,52.266,159.735
C09582=1017.954,180.165,-123.200,167.699,52.275,159.736
C09583=1017.949,179.916,-123.178,167.695,52.284,159.737
C09584=1017.943,179.667,-123.158,167.692,52.293,159.738
C09585=1017.938,179.417,-123.135,167.687,52.301,159.739
C09586=1017.934,179.168,-123.114,167.682,52.310,159.740
C09587=1017.928,178.919,-123.093,167.679,52.319,159.741
C09588=1017.923,178.671,-123.071,167.675,52.328,159.742
C09589=1017.918,178.422,-123.051,167.672,52.337,159.743
C09590=1017.913,178.173,-123.029,167.667,52.346,159.744
C09591=1017.909,177.923,-123.007,167.663,52.355,159.745
C09592=1017.903,177.675,-122.986,167.659,52.364,159.746
C09593=1017.898,177.426,-122.964,167.655,52.373,159.747
C09594=1017.893,177.176,-122.943,167.651,52.382,159.748
C09595=1017.887,176.927,-122.922,167.647,52.391,159.749
C09596=1017.883,176.678,-122.900,167.643,52.400,159.750
C09597=1017.878,176.429,-122.879,167.640,52.409,159.751
C09598=1017.873,176.180,-122.858,167.635,52.418,159.752
C09599=1017.868,175.931,-122.836,167.631,52.426,159.753
C09600=1017.863,175.682,-122.816,167.627,52.435,159.754
C09601=1017.858,175.433,-122.794,167.623,52.444,159.755
C09602=1017.853,175.184,-122.773,167.620,52.453,159.756
C09603=1017.848,174.935,-122.751,167.616,52.462,159.757
C09604=1017.843,174.686,-122.730,167.612,52.471,159.759
C09605=1017.839,174.437,-122.708,167.608,52.480,159.760
C09606=1017.833,174.188,-122.688,167.603,52.488,159.760
C09607=1017.828,173.939,-122.666,167.600,52.497,159.762
C09608=1017.823,173.690,-122.645,167.596,52.506,159.763
C09609=1017.819,173.440,-122.624,167.593,52.515,159.764
C09610=1017.814,173.192,-122.602,167.588,52.524,159.765
C09611=1017.809,172.943,-122.582,167.585,52.533,159.766
C09612=1017.804,172.694,-122.560,167.580,52.542,159.767
C09613=1017.799,172.445,-122.539,167.577,52.551,159.768
C09614=1017.794,172.195,-122.518,167.573,52.560,159.769
C09615=1017.789,171.946,-122.496,167.570,52.569,159.770
C09616=1017.784,171.697,-122.476,167.565,52.578,159.771
C09617=1017.779,171.416,-122.452,167.562,52.588,159.772
C09618=1017.773,171.135,-122.428,167.557,52.598,159.773
C09619=1017.768,170.854,-122.404,167.553,52.608,159.775
C09620=1017.762,170.573,-122.380,167.548,52.618,159.776
C09621=1017.757,170.324,-122.359,167.545,52.627,159.777
C09622=1017.753,170.075,-122.338,167.540,52.635,159.778
C09623=1017.748,169.826,-122.316,167.537,52.644,159.779
C09624=1017.743,169.577,-122.296,167.533,52.653,159.780
C09625=1017.738,169.327,-122.275,167.529,52.662,159.781
C09626=1017.733,169.079,-122.254,167.525,52.671,159.782
C09627=1017.729,168.830,-122.233,167.522,52.680,159.783
C09628=1017.724,168.581,-122.211,167.517,52.689,159.784
C09629=1017.719,168.332,-122.191,167.514,52.698,159.785
C09630=1017.714,168.082,-122.170,167.511,52.706,159.786
C09631=1017.709,167.833,-122.148,167.507,52.716,159.787
C09632=1017.704,167.584,-122.127,167.503,52.724,159.789
C09633=1017.700,167.335,-122.107,167.499,52.734,159.790
C09634=1017.695,167.086,-122.086,167.495,52.742,159.791
C09635=1017.690,166.838,-122.064,167.491,52.751,159.792
C09636=1017.686,166.588,-122.043,167.488,52.760,159.793
C09637=1017.680,166.339,-122.022,167.485,52.769,159.794
C09638=1017.676,166.090,-122.001,167.481,52.778,159.795
C09639=1017.671,165.841,-121.981,167.477,52.787,159.796
C09640=1017.667,165.592,-121.960,167.473,52.795,159.797
C09641=1017.662,165.343,-121.938,167.470,52.804,159.798
C09642=1017.657,165.094,-121.917,167.466,52.813,159.799
C09643=1017.652,164.844,-121.896,167.462,52.822,159.800
C09644=1017.648,164.596,-121.876,167.459,52.831,159.801
C09645=1017.643,164.346,-121.855,167.454,52.840,159.802
C09646=1017.638,164.097,-121.834,167.451,52.849,159.803
C09647=1017.633,163.848,-121.813,167.448,52.857,159.804
C09648=1017.629,163.599,-121.793,167.444,52.867,159.806
C09649=1017.624,163.351,-121.771,167.441,52.876,159.807
C09650=1017.619,163.101,-121.750,167.437,52.884,159.808
C09651=1017.615,162.852,-121.729,167.433,52.893,159.809
C09652=1017.610,162.603,-121.709,167.430,52.902,159.810
C09653=1017.606,162.354,-121.688,167.426,52.911,159.811
C09654=1017.600,162.105,-121.667,167.422,52.920,159.812
C09655=1017.596,161.855,-121.646,167.419,52.928,159.813
C09656=1017.591,161.607,-121.626,167.415,52.937,159.814
C09657=1017.587,161.358,-121.605,167.411,52.946,159.815
C09658=1017.582,161.108,-121.583,167.408,52.955,159.816
C09659=1017.577,160.860,-121.563,167.405,52.964,159.817
C09660=1017.573,160.610,-121.542,167.400,52.973,159.818
C09661=1017.568,160.361,-121.522,167.397,52.982,159.819
C09662=1017.563,160.112,-121.500,167.394,52.990,159.820
C09663=1017.559,159.863,-121.480,167.390,53.000,159.822
C09664=1017.554,159.614,-121.459,167.386,53.008,159.822
C09665=1017.549,159.364,-121.438,167.383,53.017,159.824
C09666=1017.545,159.116,-121.418,167.380,53.026,159.825
C09667=1017.540,158.867,-121.397,167.376,53.035,159.826
C09668=1017.536,158.617,-121.375,167.373,53.044,159.827
C09669=1017.531,158.368,-121.356,167.369,53.053,159.828
C09670=1017.526,158.119,-121.335,167.365,53.062,159.829
C09671=1017.521,157.870,-121.315,167.362,53.071,159.830
C09672=1017.516,157.621,-121.295,167.358,53.080,159.831
C09673=1017.511,157.372,-121.275,167.355,53.089,159.832
C09674=1017.506,157.123,-121.254,167.352,53.098,159.834
C09675=1017.501,156.874,-121.234,167.348,53.107,159.835
C09676=1017.497,156.624,-121.214,167.344,53.116,159.836
C09677=1017.492,156.375,-121.193,167.340,53.126,159.837
C09678=1017.487,156.126,-121.173,167.337,53.135,159.838
C09679=1017.482,155.877,-121.153,167.334,53.143,159.839
C09680=1017.477,155.628,-121.133,167.330,53.153,159.840
C09681=1017.472,155.347,-121.111,167.326,53.163,159.841
C09682=1017.467,155.065,-121.087,167.322,53.173,159.843
C09683=1017.461,154.784,-121.065,167.318,53.183,159.844
C09684=1017.456,154.503,-121.041,167.314,53.193,159.845
C09685=1017.452,154.254,-121.022,167.310,53.202,159.846
C09686=1017.446,154.004,-121.001,167.307,53.211,159.847
C09687=1017.441,153.755,-120.980,167.304,53.220,159.848
C09688=1017.437,153.506,-120.961,167.300,53.230,159.850
C09689=1017.431,153.257,-120.940,167.297,53.239,159.851
C09690=1017.427,153.008,-120.921,167.293,53.247,159.852
C09691=1017.422,152.759,-120.900,167.289,53.257,159.853
C09692=1017.417,152.509,-120.881,167.286,53.266,159.854
C09693=1017.412,152.261,-120.860,167.283,53.275,159.855
C09694=1017.407,152.011,-120.841,167.279,53.284,159.856
C09695=1017.403,151.763,-120.820,167.276,53.294,159.858
C09696=1017.398,151.513,-120.801,167.272,53.303,159.859
C09697=1017.393,151.264,-120.781,167.269,53.312,159.860
C09698=1017.388,151.015,-120.760,167.266,53.321,159.861
C09699=1017.383,150.765,-120.741,167.262,53.330,159.862
C09700=1017.378,150.517,-120.720,167.259,53.339,159.863
C09701=1017.373,150.267,-120.701,167.256,53.348,159.864
C09702=1017.369,150.018,-120.681,167.252,53.357,159.865
C09703=1017.364,149.769,-120.661,167.249,53.366,159.867
C09704=1017.360,149.520,-120.641,167.246,53.375,159.868
C09705=1017.354,149.270,-120.621,167.242,53.385,159.869
C09706=1017.350,149.021,-120.601,167.238,53.394,159.870
C09707=1017.345,148.772,-120.581,167.235,53.403,159.871
C09708=1017.340,148.523,-120.561,167.231,53.412,159.872
C09709=1017.335,148.273,-120.541,167.228,53.421,159.873
C09710=1017.330,148.025,-120.522,167.225,53.430,159.874
C09711=1017.325,147.776,-120.502,167.221,53.439,159.875
C09712=1017.321,147.527,-120.482,167.218,53.448,159.877
C09713=1017.316,147.277,-120.462,167.215,53.457,159.878
C09714=1017.311,147.028,-120.443,167.211,53.467,159.879
C09715=1017.306,146.779,-120.422,167.208,53.476,159.880
C09716=1017.302,146.530,-120.403,167.205,53.485,159.881
C09717=1017.297,146.280,-120.383,167.201,53.495,159.882
C09718=1017.292,146.031,-120.364,167.198,53.504,159.884
C09719=1017.286,145.782,-120.344,167.195,53.513,159.885
C09720=1017.282,145.533,-120.324,167.191,53.522,159.886
C09721=1017.278,145.284,-120.305,167.188,53.531,159.887
C09722=1017.273,145.034,-120.285,167.185,53.540,159.888
C09723=1017.268,144.785,-120.266,167.181,53.549,159.889
C09724=1017.263,144.536,-120.246,167.178,53.558,159.890
C09725=1017.258,144.287,-120.226,167.175,53.567,159.892
C09726=1017.252,144.038,-120.207,167.171,53.577,159.893
C09727=1017.248,143.789,-120.187,167.168,53.586,159.894
C09728=1017.243,143.539,-120.167,167.165,53.595,159.895
C09729=1017.238,143.290,-120.149,167.161,53.605,159.896
C09730=1017.234,143.041,-120.129,167.158,53.614,159.897
C09731=1017.229,142.792,-120.109,167.155,53.623,159.898
C09732=1017.224,142.543,-120.090,167.151,53.632,159.900
C09733=1017.219,142.293,-120.071,167.148,53.641,159.901
C09734=1017.214,142.044,-120.051,167.145,53.651,159.902
C09735=1017.210,141.795,-120.032,167.141,53.660,159.903
C09736=1017.204,141.546,-120.012,167.138,53.669,159.904
C09737=1017.200,141.297,-119.993,167.135,53.678,159.905
C09738=1017.195,141.047,-119.973,167.131,53.688,159.907
C09739=1017.190,140.798,-119.954,167.128,53.697,159.908
C09740=1017.186,140.549,-119.935,167.125,53.706,159.909
C09741=1017.181,140.299,-119.915,167.122,53.715,159.910
C09742=1017.176,140.051,-119.896,167.118,53.724,159.911
C09743=1017.171,139.802,-119.877,167.115,53.733,159.912
C09744=1017.166,139.552,-119.857,167.113,53.743,159.914
C09745=1017.161,139.271,-119.835,167.108,53.753,159.915
C09746=1017.155,138.990,-119.813,167.105,53.763,159.916
C09747=1017.150,138.708,-119.792,167.101,53.774,159.917
C09748=1017.144,138.426,-119.770,167.098,53.784,159.919
C09749=1017.140,138.177,-119.750,167.095,53.793,159.920
C09750=1017.135,137.929,-119.731,167.091,53.803,159.921
C09751=1017.130,137.679,-119.711,167.088,53.812,159.922
C09752=1017.125,137.430,-119.692,167.085,53.821,159.923
C09753=1017.121,137.181,-119.674,167.081,53.830,159.924
C09754=1017.115,136.931,-119.654,167.078,53.839,159.926
C09755=1017.111,136.682,-119.635,167.075,53.848,159.927
C09756=1017.106,136.433,-119.616,167.073,53.858,159.928
C09757=1017.101,136.184,-119.596,167.069,53.868,159.929
C09758=1017.096,135.934,-119.578,167.066,53.877,159.930
C09759=1017.092,135.685,-119.559,167.063,53.886,159.932
C09760=1017.087,135.436,-119.540,167.059,53.895,159.933
C09761=1017.082,135.187,-119.520,167.056,53.904,159.934
C09762=1017.077,134.937,-119.502,167.053,53.914,159.935
C09763=1017.073,134.688,-119.482,167.049,53.923,159.936
C09764=1017.067,134.439,-119.463,167.046,53.932,159.937
C09765=1017.062,134.190,-119.444,167.043,53.941,159.939
C09766=1017.058,133.941,-119.425,167.041,53.951,159.940
C09767=1017.053,133.692,-119.407,167.037,53.960,159.941
C09768=1017.048,133.442,-119.387,167.034,53.970,159.942
C09769=1017.043,133.193,-119.369,167.031,53.979,159.943
C09770=1017.038,132.944,-119.350,167.027,53.988,159.945
C09771=1017.033,132.695,-119.330,167.024,53.997,159.946
C09772=1017.028,132.445,-119.312,167.021,54.006,159.947
C09773=1017.024,132.196,-119.292,167.018,54.015,159.948
C09774=1017.019,131.947,-119.273,167.014,54.025,159.949
C09775=1017.014,131.698,-119.255,167.012,54.035,159.951
C09776=1017.010,131.449,-119.236,167.009,54.044,159.952
C09777=1017.004,131.199,-119.217,167.006,54.053,159.953
C09778=1017.000,130.950,-119.198,167.002,54.062,159.954
C09779=1016.995,130.701,-119.179,166.999,54.071,159.955
C09780=1016.990,130.452,-119.161,166.996,54.080,159.956
C09781=1016.985,130.202,-119.141,166.993,54.090,159.957
C09782=1016.980,129.952,-119.123,166.989,54.099,159.959
C09783=1016.976,129.703,-119.103,166.987,54.109,159.960
C09784=1016.971,129.454,-119.085,166.984,54.118,159.961
C09785=1016.965,129.205,-119.066,166.981,54.127,159.962
C09786=1016.961,128.955,-119.048,166.977,54.136,159.963
C09787=1016.956,128.707,-119.029,166.975,54.146,159.965
C09788=1016.951,128.457,-119.011,166.972,54.155,159.966
C09789=1016.946,128.208,-118.992,166.968,54.165,159.967
C09790=1016.941,127.959,-118.974,166.966,54.175,159.968
C09791=1016.936,127.709,-118.955,166.963,54.184,159.970
C09792=1016.931,127.460,-118.937,166.959,54.193,159.971
C09793=1016.926,127.211,-118.918,166.956,54.202,159.972
C09794=1016.921,126.962,-118.900,166.953,54.212,159.973
C09795=1016.917,126.712,-118.881,166.950,54.222,159.974
C09796=1016.912,126.463,-118.862,166.947,54.231,159.976
C09797=1016.906,126.213,-118.844,166.944,54.240,159.977
C09798=1016.902,125.964,-118.825,166.940,54.250,159.978
C09799=1016.896,125.715,-118.807,166.937,54.259,159.979
C09800=1016.892,125.466,-118.788,166.935,54.268,159.980
C09801=1016.887,125.216,-118.770,166.931,54.278,159.982
C09802=1016.882,124.968,-118.751,166.928,54.288,159.983
C09803=1016.877,124.718,-118.733,166.925,54.297,159.984
C09804=1016.872,124.469,-118.715,166.923,54.306,159.985
C09805=1016.867,124.219,-118.697,166.919,54.315,159.986
C09806=1016.862,123.970,-118.678,166.916,54.325,159.988
C09807=1016.857,123.721,-118.660,166.913,54.334,159.989
C09808=1016.852,123.471,-118.641,166.909,54.344,159.990
C09809=1016.847,123.190,-118.621,166.907,54.355,159.992
C09810=1016.841,122.909,-118.600,166.903,54.365,159.993
C09811=1016.835,122.627,-118.579,166.900,54.375,159.994
C09812=1016.830,122.346,-118.558,166.897,54.386,159.996
C09813=1016.826,122.096,-118.540,166.893,54.396,159.997
C09814=1016.821,121.847,-118.522,166.890,54.405,159.998
C09815=1016.816,121.598,-118.503,166.887,54.414,159.999
C09816=1016.811,121.349,-118.485,166.885,54.424,160.001
C09817=1016.806,121.099,-118.466,166.882,54.433,160.002
C09818=1016.801,120.850,-118.448,166.878,54.442,160.003
C09819=1016.797,120.601,-118.430,166.875,54.452,160.004
C09820=1016.792,120.352,-118.411,166.873,54.461,160.005
C09821=1016.787,120.103,-118.393,166.870,54.470,160.006
C09822=1016.782,119.853,-118.375,166.866,54.480,160.008
C09823=1016.777,119.604,-118.357,166.864,54.489,160.009
C09824=1016.772,119.355,-118.338,166.861,54.498,160.010
C09825=1016.768,119.105,-118.320,166.858,54.508,160.011
C09826=1016.763,118.857,-118.301,166.855,54.517,160.012
C09827=1016.758,118.607,-118.283,166.851,54.526,160.013
C09828=1016.753,118.358,-118.265,166.848,54.535,160.015
C09829=1016.748,118.109,-118.247,166.846,54.545,160.016
C09830=1016.743,117.859,-118.229,166.843,54.554,160.017
C09831=1016.739,117.610,-118.211,166.840,54.564,160.019
C09832=1016.734,117.360,-118.192,166.837,54.573,160.020
C09833=1016.729,117.111,-118.174,166.834,54.582,160.021
C09834=1016.724,116.862,-118.156,166.831,54.591,160.022
C09835=1016.719,116.613,-118.137,166.828,54.601,160.023
C09836=1016.714,116.364,-118.119,166.825,54.610,160.024
C09837=1016.710,116.114,-118.101,166.823,54.619,160.026
C09838=1016.705,115.865,-118.083,166.820,54.629,160.027
C09839=1016.700,115.616,-118.065,166.816,54.638,160.028
C09840=1016.695,115.366,-118.046,166.814,54.648,160.029
C09841=1016.691,115.117,-118.028,166.811,54.657,160.030
C09842=1016.687,114.867,-118.010,166.808,54.666,160.032
C09843=1016.682,114.618,-117.991,166.805,54.675,160.033
C09844=1016.677,114.369,-117.973,166.802,54.684,160.034
C09845=1016.672,114.119,-117.955,166.800,54.693,160.035
C09846=1016.667,113.870,-117.937,166.796,54.703,160.036
C09847=1016.663,113.620,-117.919,166.793,54.712,160.038
C09848=1016.658,113.371,-117.901,166.790,54.721,160.039
C09849=1016.654,113.122,-117.883,166.788,54.731,160.040
C09850=1016.649,112.873,-117.865,166.785,54.740,160.041
C09851=1016.644,112.624,-117.846,166.782,54.749,160.042
C09852=1016.639,112.374,-117.828,166.779,54.758,160.044
C09853=1016.635,112.125,-117.810,166.776,54.767,160.045
C09854=1016.630,111.876,-117.792,166.774,54.777,160.046
C09855=1016.624,111.627,-117.774,166.770,54.787,160.047
C09856=1016.620,111.377,-117.757,166.768,54.796,160.049
C09857=1016.615,111.127,-117.739,166.765,54.805,160.050
C09858=1016.610,110.878,-117.721,166.762,54.814,160.051
C09859=1016.605,110.629,-117.703,166.759,54.824,160.052
C09860=1016.600,110.380,-117.685,166.756,54.833,160.053
C09861=1016.596,110.130,-117.668,166.753,54.843,160.055
C09862=1016.591,109.881,-117.650,166.751,54.852,160.056
C09863=1016.586,109.632,-117.632,166.748,54.862,160.057
C09864=1016.581,109.383,-117.614,166.745,54.871,160.058
C09865=1016.576,109.133,-117.597,166.741,54.880,160.059
C09866=1016.571,108.884,-117.579,166.739,54.890,160.061
C09867=1016.566,108.634,-117.561,166.736,54.900,160.062
C09868=1016.561,108.385,-117.544,166.734,54.909,160.063
C09869=1016.557,108.136,-117.526,166.730,54.918,160.064
C09870=1016.551,107.887,-117.509,166.728,54.928,160.066
C09871=1016.547,107.637,-117.491,166.725,54.938,160.067
C09872=1016.541,107.388,-117.474,166.722,54.947,160.068
C09873=1016.536,107.106,-117.454,166.719,54.957,160.070
C09874=1016.530,106.825,-117.434,166.715,54.969,160.071
C09875=1016.525,106.543,-117.414,166.712,54.979,160.072
C09876=1016.519,106.263,-117.395,166.709,54.990,160.074
C09877=1016.515,106.013,-117.377,166.706,54.999,160.075
C09878=1016.510,105.763,-117.359,166.704,55.008,160.076
C09879=1016.505,105.514,-117.342,166.701,55.018,160.077
C09880=1016.500,105.265,-117.323,166.697,55.027,160.079
C09881=1016.495,105.016,-117.307,166.695,55.036,160.080
C09882=1016.490,104.767,-117.289,166.692,55.046,160.081
C09883=1016.485,104.517,-117.272,166.690,55.056,160.082
C09884=1016.480,104.268,-117.254,166.687,55.065,160.084
C09885=1016.475,104.018,-117.237,166.684,55.074,160.085
C09886=1016.471,103.769,-117.219,166.681,55.084,160.086
C09887=1016.466,103.520,-117.202,166.678,55.093,160.087
C09888=1016.461,103.270,-117.184,166.676,55.103,160.089
C09889=1016.456,103.021,-117.167,166.673,55.112,160.090
C09890=1016.451,102.771,-117.149,166.670,55.121,160.091
C09891=1016.446,102.523,-117.132,166.668,55.131,160.092
C09892=1016.442,102.273,-117.114,166.664,55.140,160.093
C09893=1016.437,102.024,-117.096,166.661,55.150,160.095
C09894=1016.432,101.774,-117.079,166.659,55.159,160.096
C09895=1016.427,101.525,-117.062,166.656,55.168,160.097
C09896=1016.422,101.276,-117.045,166.653,55.177,160.098
C09897=1016.417,101.026,-117.027,166.651,55.187,160.100
C09898=1016.412,100.777,-117.010,166.648,55.197,160.101
C09899=1016.408,100.528,-116.992,166.645,55.206,160.102
C09900=1016.403,100.278,-116.975,166.642,55.216,160.103
C09901=1016.398,100.028,-116.958,166.639,55.225,160.104
C09902=1016.393,99.779,-116.940,166.637,55.234,160.106
C09903=1016.389,99.530,-116.923,166.634,55.243,160.107
C09904=1016.383,99.281,-116.905,166.631,55.253,160.108
C09905=1016.379,99.031,-116.888,166.629,55.262,160.109
C09906=1016.374,98.782,-116.872,166.626,55.271,160.111
C09907=1016.369,98.533,-116.854,166.622,55.281,160.112
C09908=1016.364,98.283,-116.837,166.620,55.291,160.113
C09909=1016.359,98.033,-116.820,166.618,55.300,160.114
C09910=1016.354,97.785,-116.802,166.615,55.309,160.116
C09911=1016.349,97.535,-116.786,166.612,55.319,160.117
C09912=1016.345,97.285,-116.768,166.609,55.329,160.118
C09913=1016.340,97.036,-116.752,166.607,55.338,160.119
C09914=1016.334,96.787,-116.734,166.604,55.348,160.121
C09915=1016.329,96.538,-116.717,166.601,55.357,160.122
C09916=1016.325,96.288,-116.700,166.599,55.366,160.123
C09917=1016.320,96.039,-116.683,166.595,55.376,160.124
C09918=1016.315,95.789,-116.666,166.593,55.386,160.126
C09919=1016.309,95.540,-116.649,166.590,55.395,160.127
C09920=1016.305,95.291,-116.632,166.588,55.405,160.128
C09921=1016.300,95.041,-116.615,166.585,55.414,160.129
C09922=1016.295,94.791,-116.598,166.582,55.423,160.131
C09923=1016.291,94.543,-116.582,166.579,55.433,160.132
C09924=1016.285,94.293,-116.564,166.576,55.442,160.133
C09925=1016.281,94.044,-116.547,166.574,55.452,160.134
C09926=1016.276,93.795,-116.530,166.571,55.461,160.136
C09927=1016.271,93.545,-116.513,166.569,55.471,160.137
C09928=1016.266,93.296,-116.497,166.566,55.480,160.138
C09929=1016.261,93.046,-116.480,166.564,55.489,160.139
C09930=1016.256,92.797,-116.462,166.560,55.499,160.140
C09931=1016.251,92.548,-116.445,166.557,55.508,160.142
C09932=1016.246,92.298,-116.428,166.555,55.518,160.143
C09933=1016.241,92.049,-116.412,166.552,55.527,160.144
C09934=1016.237,91.799,-116.395,166.550,55.536,160.145
C09935=1016.232,91.550,-116.378,166.547,55.546,160.147
C09936=1016.227,91.301,-116.361,166.544,55.555,160.148
C09937=1016.221,91.019,-116.342,166.542,55.566,160.149
C09938=1016.216,90.738,-116.323,166.539,55.577,160.151
C09939=1016.210,90.457,-116.304,166.536,55.587,160.152
C09940=1016.205,90.176,-116.285,166.533,55.597,160.153
C09941=1016.201,89.927,-116.268,166.530,55.607,160.155
C09942=1016.196,89.677,-116.251,166.526,55.616,160.156
C09943=1016.191,89.428,-116.234,166.524,55.626,160.157
C09944=1016.186,89.179,-116.217,166.521,55.635,160.158
C09945=1016.181,88.929,-116.201,166.519,55.644,160.159
C09946=1016.177,88.680,-116.183,166.516,55.654,160.161
C09947=1016.171,88.430,-116.167,166.514,55.663,160.162
C09948=1016.166,88.181,-116.150,166.512,55.673,160.163
C09949=1016.161,87.932,-116.134,166.509,55.683,160.165
C09950=1016.156,87.682,-116.117,166.505,55.692,160.166
C09951=1016.151,87.433,-116.101,166.503,55.702,160.167
C09952=1016.146,87.183,-116.084,166.500,55.711,160.168
C09953=1016.142,86.934,-116.068,166.498,55.720,160.169
C09954=1016.137,86.684,-116.051,166.496,55.730,160.171
C09955=1016.132,86.435,-116.035,166.492,55.740,160.172
C09956=1016.127,86.186,-116.018,166.490,55.749,160.173
C09957=1016.122,85.936,-116.001,166.487,55.759,160.175
C09958=1016.116,85.687,-115.986,166.484,55.768,160.176
C09959=1016.111,85.437,-115.969,166.482,55.777,160.177
C09960=1016.107,85.188,-115.952,166.479,55.787,160.178
C09961=1016.101,84.938,-115.935,166.476,55.797,160.179
C09962=1016.097,84.689,-115.919,166.474,55.807,160.181
C09963=1016.092,84.440,-115.902,166.471,55.816,160.182
C09964=1016.087,84.190,-115.886,166.469,55.825,160.183
C09965=1016.082,83.940,-115.870,166.466,55.835,160.185
C09966=1016.077,83.692,-115.853,166.464,55.844,160.186
C09967=1016.072,83.442,-115.836,166.461,55.853,160.187
C09968=1016.067,83.193,-115.821,166.458,55.863,160.188
C09969=1016.062,82.943,-115.804,166.455,55.873,160.189
C09970=1016.057,82.694,-115.788,166.453,55.882,160.191
C09971=1016.052,82.444,-115.771,166.450,55.891,160.192
C09972=1016.048,82.195,-115.754,166.448,55.901,160.193
C09973=1016.043,81.945,-115.738,166.445,55.910,160.195
C09974=1016.038,81.696,-115.722,166.443,55.919,160.196
C09975=1016.033,81.447,-115.705,166.440,55.929,160.197
C09976=1016.029,81.197,-115.689,166.438,55.938,160.198
C09977=1016.023,80.948,-115.673,166.434,55.948,160.199
C09978=1016.018,80.699,-115.656,166.432,55.957,160.201
C09979=1016.013,80.450,-115.640,166.429,55.967,160.202
C09980=1016.008,80.199,-115.624,166.427,55.976,160.203
C09981=1016.004,79.950,-115.607,166.424,55.985,160.204
C09982=1015.999,79.701,-115.590,166.422,55.995,160.206
C09983=1015.994,79.451,-115.575,166.419,56.004,160.207
C09984=1015.990,79.202,-115.558,166.417,56.014,160.208
C09985=1015.984,78.953,-115.541,166.414,56.023,160.209
C09986=1015.980,78.704,-115.525,166.412,56.032,160.211
C09987=1015.974,78.454,-115.509,166.409,56.042,160.212
C09988=1015.970,78.205,-115.493,166.407,56.051,160.213
C09989=1015.964,77.955,-115.476,166.404,56.060,160.214
C09990=1015.960,77.705,-115.460,166.401,56.069,160.215
C09991=1015.955,77.456,-115.444,166.399,56.079,160.217
C09992=1015.951,77.206,-115.428,166.396,56.088,160.218
C09993=1015.946,76.957,-115.411,166.394,56.097,160.219
C09994=1015.940,76.708,-115.395,166.390,56.107,160.220
C09995=1015.936,76.458,-115.379,166.388,56.117,160.222
C09996=1015.931,76.209,-115.363,166.386,56.126,160.223
//INST
///DATE 2021/06/17 10:59
///ATTR SC,RW,RJ
////FRAME ROBOT
///GROUP1 RB1
NOP
MOVL C00000 V=800.0 PL=0
MOVL C00001 V=800.0 PL=0
MOVL C00002 V=800.0 PL=0
MOVL C00003 V=800.0 PL=0
MOVL C00004 V=800.0 PL=0
MOVL C00005 V=800.0 PL=0
MOVL C00006 V=800.0 PL=0
MOVL C00007 V=800.0 PL=0
MOVL C00008 V=800.0 PL=0
MOVL C00009 V=800.0 PL=0
MOVL C00010 V=800.0 PL=0
MOVL C00011 V=800.0 PL=0
MOVL C00012 V=800.0 PL=0
MOVL C00013 V=800.0 PL=0
MOVL C00014 V=800.0 PL=0
MOVL C00015 V=800.0 PL=0
MOVL C00016 V=800.0 PL=0
MOVL C00017 V=800.0 PL=0
MOVL C00018 V=800.0 PL=0
MOVL C00019 V=800.0 PL=0
MOVL C00020 V=800.0 PL=0
MOVL C00021 V=800.0 PL=0
MOVL C00022 V=800.0 PL=0
MOVL C00023 V=800.0 PL=0
MOVL C00024 V=800.0 PL=0
MOVL C00025 V=800.0 PL=0
MOVL C00026 V=800.0 PL=0
MOVL C00027 V=800.0 PL=0
MOVL C00028 V=800.0 PL=0
MOVL C00029 V=800.0 PL=0
MOVL C00030 V=800.0 PL=0
MOVL C00031 V=800.0 PL=0
MOVL C00032 V=800.0 PL=0
MOVL C00033 V=800.0 PL=0
MOVL C00034 V=800.0 PL=0
MOVL C00035 V=800.0 PL=0
MOVL C00036 V=800.0 PL=0
MOVL C00037 V=800.0 PL=0
MOVL C00038 V=800.0 PL=0
MOVL C00039 V=800.0 PL=0
MOVL C00040 V=800.0 PL=0
MOVL C00041 V=800.0 PL=0
MOVL C00042 V=800.0 PL=0
MOVL C00043 V=800.0 PL=0
MOVL C00044 V=800.0 PL=0
MOVL C00045 V=800.0 PL=0
MOVL C00046 V=800.0 PL=0
MOVL C00047 V=800.0 PL=0
MOVL C00048 V=800.0 PL=0
MOVL C00049 V=800.0 PL=0
MOVL C00050 V=800.0 PL=0
MOVL C00051 V=800.0 PL=0
MOVL C00052 V=800.0 PL=0
MOVL C00053 V=800.0 PL=0
MOVL C00054 V=800.0 PL=0
MOVL C00055 V=800.0 PL=0
MOVL C00056 V=800.0 PL=0
MOVL C00057 V=800.0 PL=0
MOVL C00058 V=800.0 PL=0
MOVL C00059 V=800.0 PL=0
MOVL C00060 V=800.0 PL=0
MOVL C00061 V=800.0 PL=0
MOVL C00062 V=800.0 PL=0
MOVL C00063 V=800.0 PL=0
MOVL C00064 V=800.0 PL=0
MOVL C00065 V=800.0 PL=0
MOVL C00066 V=800.0 PL=0
MOVL C00067 V=800.0 PL=0
MOVL C00068 V=800.0 PL=0
MOVL C00069 V=800.0 PL=0
MOVL C00070 V=800.0 PL=0
MOVL C00071 V=800.0 PL=0
MOVL C00072 V=800.0 PL=0
MOVL C00073 V=800.0 PL=0
MOVL C00074 V=800.0 PL=0
MOVL C00075 V=800.0 PL=0
MOVL C00076 V=800.0 PL=0
MOVL C00077 V=800.0 PL=0
MOVL C00078 V=800.0 PL=0
MOVL C00079 V=800.0 PL=0
MOVL C00080 V=800.0 PL=0
MOVL C00081 V=800.0 PL=0
MOVL C00082 V=800.0 PL=0
MOVL C00083 V=800.0 PL=0
MOVL C00084 V=800.0 PL=0
MOVL C00085 V=800.0 PL=0
MOVL C00086 V=800.0 PL=0
MOVL C00087 V=800.0 PL=0
MOVL C00088 V=800.0 PL=0
MOVL C00089 V=800.0 PL=0
MOVL C00090 V=800.0 PL=0
MOVL C00091 V=800.0 PL=0
MOVL C00092 V=800.0 PL=0
MOVL C00093 V=800.0 PL=0
MOVL C00094 V=800.0 PL=0
MOVL C00095 V=800.0 PL=0
MOVL C00096 V=800.0 PL=0
MOVL C00097 V=800.0 PL=0
MOVL C00098 V=800.0 PL=0
MOVL C00099 V=800.0 PL=0
MOVL C00100 V=800.0 PL=0
MOVL C00101 V=800.0 PL=0
MOVL C00102 V=800.0 PL=0
MOVL C00103 V=800.0 PL=0
MOVL C00104 V=800.0 PL=0
MOVL C00105 V=800.0 PL=0
MOVL C00106 V=800.0 PL=0
MOVL C00107 V=800.0 PL=0
MOVL C00108 V=800.0 PL=0
MOVL C00109 V=800.0 PL=0
MOVL C00110 V=800.0 PL=0
MOVL C00111 V=800.0 PL=0
MOVL C00112 V=800.0 PL=0
MOVL C00113 V=800.0 PL=0
MOVL C00114 V=800.0 PL=0
MOVL C00115 V=800.0 PL=0
MOVL C00116 V=800.0 PL=0
MOVL C00117 V=800.0 PL=0
MOVL C00118 V=800.0 PL=0
MOVL C00119 V=800.0 PL=0
MOVL C00120 V=800.0 PL=0
MOVL C00121 V=800.0 PL=0
MOVL C00122 V=800.0 PL=0
MOVL C00123 V=800.0 PL=0
MOVL C00124 V=800.0 PL=0
MOVL C00125 V=800.0 PL=0
MOVL C00126 V=800.0 PL=0
MOVL C00127 V=800.0 PL=0
MOVL C00128 V=800.0 PL=0
MOVL C00129 V=800.0 PL=0
MOVL C00130 V=800.0 PL=0
MOVL C00131 V=800.0 PL=0
MOVL C00132 V=800.0 PL=0
MOVL C00133 V=800.0 PL=0
MOVL C00134 V=800.0 PL=0
MOVL C00135 V=800.0 PL=0
MOVL C00136 V=800.0 PL=0
MOVL C00137 V=800.0 PL=0
MOVL C00138 V=800.0 PL=0
MOVL C00139 V=800.0 PL=0
MOVL C00140 V=800.0 PL=0
MOVL C00141 V=800.0 PL=0
MOVL C00142 V=800.0 PL=0
MOVL C00143 V=800.0 PL=0
MOVL C00144 V=800.0 PL=0
MOVL C00145 V=800.0 PL=0
MOVL C00146 V=800.0 PL=0
MOVL C00147 V=800.0 PL=0
MOVL C00148 V=800.0 PL=0
MOVL C00149 V=800.0 PL=0
MOVL C00150 V=800.0 PL=0
MOVL C00151 V=800.0 PL=0
MOVL C00152 V=800.0 PL=0
MOVL C00153 V=800.0 PL=0
MOVL C00154 V=800.0 PL=0
MOVL C00155 V=800.0 PL=0
MOVL C00156 V=800.0 PL=0
MOVL C00157 V=800.0 PL=0
MOVL C00158 V=800.0 PL=0
MOVL C00159 V=800.0 PL=0
MOVL C00160 V=800.0 PL=0
MOVL C00161 V=800.0 PL=0
MOVL C00162 V=800.0 PL=0
MOVL C00163 V=800.0 PL=0
MOVL C00164 V=800.0 PL=0
MOVL C00165 V=800.0 PL=0
MOVL C00166 V=800.0 PL=0
MOVL C00167 V=800.0 PL=0
MOVL C00168 V=800.0 PL=0
MOVL C00169 V=800.0 PL=0
MOVL C00170 V=800.0 PL=0
MOVL C00171 V=800.0 PL=0
MOVL C00172 V=800.0 PL=0
MOVL C00173 V=800.0 PL=0
MOVL C00174 V=800.0 PL=0
MOVL C00175 V=800.0 PL=0
MOVL C00176 V=800.0 PL=0
MOVL C00177 V=800.0 PL=0
MOVL C00178 V=800.0 PL=0
MOVL C00179 V=800.0 PL=0
MOVL C00180 V=800.0 PL=0
MOVL C00181 V=800.0 PL=0
MOVL C00182 V=800.0 PL=0
MOVL C00183 V=800.0 PL=0
MOVL C00184 V=800.0 PL=0
MOVL C00185 V=800.0 PL=0
MOVL C00186 V=800.0 PL=0
MOVL C00187 V=800.0 PL=0
MOVL C00188 V=800.0 PL=0
MOVL C00189 V=800.0 PL=0
MOVL C00190 V=800.0 PL=0
MOVL C00191 V=800.0 PL=0
MOVL C00192 V=800.0 PL=0
MOVL C00193 V=800.0 PL=0
MOVL C00194 V=800.0 PL=0
MOVL C00195 V=800.0 PL=0
MOVL C00196 V=800.0 PL=0
MOVL C00197 V=800.0 PL=0
MOVL C00198 V=800.0 PL=0
MOVL C00199 V=800.0 PL=0
MOVL C00200 V=800.0 PL=0
MOVL C00201 V=800.0 PL=0
MOVL C00202 V=800.0 PL=0
MOVL C00203 V=800.0 PL=0
MOVL C00204 V=800.0 PL=0
MOVL C00205 V=800.0 PL=0
MOVL C00206 V=800.0 PL=0
MOVL C00207 V=800.0 PL=0
MOVL C00208 V=800.0 PL=0
MOVL C00209 V=800.0 PL=0
MOVL C00210 V=800.0 PL=0
MOVL C00211 V=800.0 PL=0
MOVL C00212 V=800.0 PL=0
MOVL C00213 V=800.0 PL=0
MOVL C00214 V=800.0 PL=0
MOVL C00215 V=800.0 PL=0
MOVL C00216 V=800.0 PL=0
MOVL C00217 V=800.0 PL=0
MOVL C00218 V=800.0 PL=0
MOVL C00219 V=800.0 PL=0
MOVL C00220 V=800.0 PL=0
MOVL C00221 V=800.0 PL=0
MOVL C00222 V=800.0 PL=0
MOVL C00223 V=800.0 PL=0
MOVL C00224 V=800.0 PL=0
MOVL C00225 V=800.0 PL=0
MOVL C00226 V=800.0 PL=0
MOVL C00227 V=800.0 PL=0
MOVL C00228 V=800.0 PL=0
MOVL C00229 V=800.0 PL=0
MOVL C00230 V=800.0 PL=0
MOVL C00231 V=800.0 PL=0
MOVL C00232 V=800.0 PL=0
MOVL C00233 V=800.0 PL=0
MOVL C00234 V=800.0 PL=0
MOVL C00235 V=800.0 PL=0
MOVL C00236 V=800.0 PL=0
MOVL C00237 V=800.0 PL=0
MOVL C00238 V=800.0 PL=0
MOVL C00239 V=800.0 PL=0
MOVL C00240 V=800.0 PL=0
MOVL C00241 V=800.0 PL=0
MOVL C00242 V=800.0 PL=0
MOVL C00243 V=800.0 PL=0
MOVL C00244 V=800.0 PL=0
MOVL C00245 V=800.0 PL=0
MOVL C00246 V=800.0 PL=0
MOVL C00247 V=800.0 PL=0
MOVL C00248 V=800.0 PL=0
MOVL C00249 V=800.0 PL=0
MOVL C00250 V=800.0 PL=0
MOVL C00251 V=800.0 PL=0
MOVL C00252 V=800.0 PL=0
MOVL C00253 V=800.0 PL=0
MOVL C00254 V=800.0 PL=0
MOVL C00255 V=800.0 PL=0
MOVL C00256 V=800.0 PL=0
MOVL C00257 V=800.0 PL=0
MOVL C00258 V=800.0 PL=0
MOVL C00259 V=800.0 PL=0
MOVL C00260 V=800.0 PL=0
MOVL C00261 V=800.0 PL=0
MOVL C00262 V=800.0 PL=0
MOVL C00263 V=800.0 PL=0
MOVL C00264 V=800.0 PL=0
MOVL C00265 V=800.0 PL=0
MOVL C00266 V=800.0 PL=0
MOVL C00267 V=800.0 PL=0
MOVL C00268 V=800.0 PL=0
MOVL C00269 V=800.0 PL=0
MOVL C00270 V=800.0 PL=0
MOVL C00271 V=800.0 PL=0
MOVL C00272 V=800.0 PL=0
MOVL C00273 V=800.0 PL=0
MOVL C00274 V=800.0 PL=0
MOVL C00275 V=800.0 PL=0
MOVL C00276 V=800.0 PL=0
MOVL C00277 V=800.0 PL=0
MOVL C00278 V=800.0 PL=0
MOVL C00279 V=800.0 PL=0
MOVL C00280 V=800.0 PL=0
MOVL C00281 V=800.0 PL=0
MOVL C00282 V=800.0 PL=0
MOVL C00283 V=800.0 PL=0
MOVL C00284 V=800.0 PL=0
MOVL C00285 V=800.0 PL=0
MOVL C00286 V=800.0 PL=0
MOVL C00287 V=800.0 PL=0
MOVL C00288 V=800.0 PL=0
MOVL C00289 V=800.0 PL=0
MOVL C00290 V=800.0 PL=0
MOVL C00291 V=800.0 PL=0
MOVL C00292 V=800.0 PL=0
MOVL C00293 V=800.0 PL=0
MOVL C00294 V=800.0 PL=0
MOVL C00295 V=800.0 PL=0
MOVL C00296 V=800.0 PL=0
MOVL C00297 V=800.0 PL=0
MOVL C00298 V=800.0 PL=0
MOVL C00299 V=800.0 PL=0
MOVL C00300 V=800.0 PL=0
MOVL C00301 V=800.0 PL=0
MOVL C00302 V=800.0 PL=0
MOVL C00303 V=800.0 PL=0
MOVL C00304 V=800.0 PL=0
MOVL C00305 V=800.0 PL=0
MOVL C00306 V=800.0 PL=0
MOVL C00307 V=800.0 PL=0
MOVL C00308 V=800.0 PL=0
MOVL C00309 V=800.0 PL=0
MOVL C00310 V=800.0 PL=0
MOVL C00311 V=800.0 PL=0
MOVL C00312 V=800.0 PL=0
MOVL C00313 V=800.0 PL=0
MOVL C00314 V=800.0 PL=0
MOVL C00315 V=800.0 PL=0
MOVL C00316 V=800.0 PL=0
MOVL C00317 V=800.0 PL=0
MOVL C00318 V=800.0 PL=0
MOVL C00319 V=800.0 PL=0
MOVL C00320 V=800.0 PL=0
MOVL C00321 V=800.0 PL=0
MOVL C00322 V=800.0 PL=0
MOVL C00323 V=800.0 PL=0
MOVL C00324 V=800.0 PL=0
MOVL C00325 V=800.0 PL=0
MOVL C00326 V=800.0 PL=0
MOVL C00327 V=800.0 PL=0
MOVL C00328 V=800.0 PL=0
MOVL C00329 V=800.0 PL=0
MOVL C00330 V=800.0 PL=0
MOVL C00331 V=800.0 PL=0
MOVL C00332 V=800.0 PL=0
MOVL C00333 V=800.0 PL=0
MOVL C00334 V=800.0 PL=0
MOVL C00335 V=800.0 PL=0
MOVL C00336 V=800.0 PL=0
MOVL C00337 V=800.0 PL=0
MOVL C00338 V=800.0 PL=0
MOVL C00339 V=800.0 PL=0
MOVL C00340 V=800.0 PL=0
MOVL C00341 V=800.0 PL=0
MOVL C00342 V=800.0 PL=0
MOVL C00343 V=800.0 PL=0
MOVL C00344 V=800.0 PL=0
MOVL C00345 V=800.0 PL=0
MOVL C00346 V=800.0 PL=0
MOVL C00347 V=800.0 PL=0
MOVL C00348 V=800.0 PL=0
MOVL C00349 V=800.0 PL=0
MOVL C00350 V=800.0 PL=0
MOVL C00351 V=800.0 PL=0
MOVL C00352 V=800.0 PL=0
MOVL C00353 V=800.0 PL=0
MOVL C00354 V=800.0 PL=0
MOVL C00355 V=800.0 PL=0
MOVL C00356 V=800.0 PL=0
MOVL C00357 V=800.0 PL=0
MOVL C00358 V=800.0 PL=0
MOVL C00359 V=800.0 PL=0
MOVL C00360 V=800.0 PL=0
MOVL C00361 V=800.0 PL=0
MOVL C00362 V=800.0 PL=0
MOVL C00363 V=800.0 PL=0
MOVL C00364 V=800.0 PL=0
MOVL C00365 V=800.0 PL=0
MOVL C00366 V=800.0 PL=0
MOVL C00367 V=800.0 PL=0
MOVL C00368 V=800.0 PL=0
MOVL C00369 V=800.0 PL=0
MOVL C00370 V=800.0 PL=0
MOVL C00371 V=800.0 PL=0
MOVL C00372 V=800.0 PL=0
MOVL C00373 V=800.0 PL=0
MOVL C00374 V=800.0 PL=0
MOVL C00375 V=800.0 PL=0
MOVL C00376 V=800.0 PL=0
MOVL C00377 V=800.0 PL=0
MOVL C00378 V=800.0 PL=0
MOVL C00379 V=800.0 PL=0
MOVL C00380 V=800.0 PL=0
MOVL C00381 V=800.0 PL=0
MOVL C00382 V=800.0 PL=0
MOVL C00383 V=800.0 PL=0
MOVL C00384 V=800.0 PL=0
MOVL C00385 V=800.0 PL=0
MOVL C00386 V=800.0 PL=0
MOVL C00387 V=800.0 PL=0
MOVL C00388 V=800.0 PL=0
MOVL C00389 V=800.0 PL=0
MOVL C00390 V=800.0 PL=0
MOVL C00391 V=800.0 PL=0
MOVL C00392 V=800.0 PL=0
MOVL C00393 V=800.0 PL=0
MOVL C00394 V=800.0 PL=0
MOVL C00395 V=800.0 PL=0
MOVL C00396 V=800.0 PL=0
MOVL C00397 V=800.0 PL=0
MOVL C00398 V=800.0 PL=0
MOVL C00399 V=800.0 PL=0
MOVL C00400 V=800.0 PL=0
MOVL C00401 V=800.0 PL=0
MOVL C00402 V=800.0 PL=0
MOVL C00403 V=800.0 PL=0
MOVL C00404 V=800.0 PL=0
MOVL C00405 V=800.0 PL=0
MOVL C00406 V=800.0 PL=0
MOVL C00407 V=800.0 PL=0
MOVL C00408 V=800.0 PL=0
MOVL C00409 V=800.0 PL=0
MOVL C00410 V=800.0 PL=0
MOVL C00411 V=800.0 PL=0
MOVL C00412 V=800.0 PL=0
MOVL C00413 V=800.0 PL=0
MOVL C00414 V=800.0 PL=0
MOVL C00415 V=800.0 PL=0
MOVL C00416 V=800.0 PL=0
MOVL C00417 V=800.0 PL=0
MOVL C00418 V=800.0 PL=0
MOVL C00419 V=800.0 PL=0
MOVL C00420 V=800.0 PL=0
MOVL C00421 V=800.0 PL=0
MOVL C00422 V=800.0 PL=0
MOVL C00423 V=800.0 PL=0
MOVL C00424 V=800.0 PL=0
MOVL C00425 V=800.0 PL=0
MOVL C00426 V=800.0 PL=0
MOVL C00427 V=800.0 PL=0
MOVL C00428 V=800.0 PL=0
MOVL C00429 V=800.0 PL=0
MOVL C00430 V=800.0 PL=0
MOVL C00431 V=800.0 PL=0
MOVL C00432 V=800.0 PL=0
MOVL C00433 V=800.0 PL=0
MOVL C00434 V=800.0 PL=0
MOVL C00435 V=800.0 PL=0
MOVL C00436 V=800.0 PL=0
MOVL C00437 V=800.0 PL=0
MOVL C00438 V=800.0 PL=0
MOVL C00439 V=800.0 PL=0
MOVL C00440 V=800.0 PL=0
MOVL C00441 V=800.0 PL=0
MOVL C00442 V=800.0 PL=0
MOVL C00443 V=800.0 PL=0
MOVL C00444 V=800.0 PL=0
MOVL C00445 V=800.0 PL=0
MOVL C00446 V=800.0 PL=0
MOVL C00447 V=800.0 PL=0
MOVL C00448 V=800.0 PL=0
MOVL C00449 V=800.0 PL=0
MOVL C00450 V=800.0 PL=0
MOVL C00451 V=800.0 PL=0
MOVL C00452 V=800.0 PL=0
MOVL C00453 V=800.0 PL=0
MOVL C00454 V=800.0 PL=0
MOVL C00455 V=800.0 PL=0
MOVL C00456 V=800.0 PL=0
MOVL C00457 V=800.0 PL=0
MOVL C00458 V=800.0 PL=0
MOVL C00459 V=800.0 PL=0
MOVL C00460 V=800.0 PL=0
MOVL C00461 V=800.0 PL=0
MOVL C00462 V=800.0 PL=0
MOVL C00463 V=800.0 PL=0
MOVL C00464 V=800.0 PL=0
MOVL C00465 V=800.0 PL=0
MOVL C00466 V=800.0 PL=0
MOVL C00467 V=800.0 PL=0
MOVL C00468 V=800.0 PL=0
MOVL C00469 V=800.0 PL=0
MOVL C00470 V=800.0 PL=0
MOVL C00471 V=800.0 PL=0
MOVL C00472 V=800.0 PL=0
MOVL C00473 V=800.0 PL=0
MOVL C00474 V=800.0 PL=0
MOVL C00475 V=800.0 PL=0
MOVL C00476 V=800.0 PL=0
MOVL C00477 V=800.0 PL=0
MOVL C00478 V=800.0 PL=0
MOVL C00479 V=800.0 PL=0
MOVL C00480 V=800.0 PL=0
MOVL C00481 V=800.0 PL=0
MOVL C00482 V=800.0 PL=0
MOVL C00483 V=800.0 PL=0
MOVL C00484 V=800.0 PL=0
MOVL C00485 V=800.0 PL=0
MOVL C00486 V=800.0 PL=0
MOVL C00487 V=800.0 PL=0
MOVL C00488 V=800.0 PL=0
MOVL C00489 V=800.0 PL=0
MOVL C00490 V=800.0 PL=0
MOVL C00491 V=800.0 PL=0
MOVL C00492 V=800.0 PL=0
MOVL C00493 V=800.0 PL=0
MOVL C00494 V=800.0 PL=0
MOVL C00495 V=800.0 PL=0
MOVL C00496 V=800.0 PL=0
MOVL C00497 V=800.0 PL=0
MOVL C00498 V=800.0 PL=0
MOVL C00499 V=800.0 PL=0
MOVL C00500 V=800.0 PL=0
MOVL C00501 V=800.0 PL=0
MOVL C00502 V=800.0 PL=0
MOVL C00503 V=800.0 PL=0
MOVL C00504 V=800.0 PL=0
MOVL C00505 V=800.0 PL=0
MOVL C00506 V=800.0 PL=0
MOVL C00507 V=800.0 PL=0
MOVL C00508 V=800.0 PL=0
MOVL C00509 V=800.0 PL=0
MOVL C00510 V=800.0 PL=0
MOVL C00511 V=800.0 PL=0
MOVL C00512 V=800.0 PL=0
MOVL C00513 V=800.0 PL=0
MOVL C00514 V=800.0 PL=0
MOVL C00515 V=800.0 PL=0
MOVL C00516 V=800.0 PL=0
MOVL C00517 V=800.0 PL=0
MOVL C00518 V=800.0 PL=0
MOVL C00519 V=800.0 PL=0
MOVL C00520 V=800.0 PL=0
MOVL C00521 V=800.0 PL=0
MOVL C00522 V=800.0 PL=0
MOVL C00523 V=800.0 PL=0
MOVL C00524 V=800.0 PL=0
MOVL C00525 V=800.0 PL=0
MOVL C00526 V=800.0 PL=0
MOVL C00527 V=800.0 PL=0
MOVL C00528 V=800.0 PL=0
MOVL C00529 V=800.0 PL=0
MOVL C00530 V=800.0 PL=0
MOVL C00531 V=800.0 PL=0
MOVL C00532 V=800.0 PL=0
MOVL C00533 V=800.0 PL=0
MOVL C00534 V=800.0 PL=0
MOVL C00535 V=800.0 PL=0
MOVL C00536 V=800.0 PL=0
MOVL C00537 V=800.0 PL=0
MOVL C00538 V=800.0 PL=0
MOVL C00539 V=800.0 PL=0
MOVL C00540 V=800.0 PL=0
MOVL C00541 V=800.0 PL=0
MOVL C00542 V=800.0 PL=0
MOVL C00543 V=800.0 PL=0
MOVL C00544 V=800.0 PL=0
MOVL C00545 V=800.0 PL=0
MOVL C00546 V=800.0 PL=0
MOVL C00547 V=800.0 PL=0
MOVL C00548 V=800.0 PL=0
MOVL C00549 V=800.0 PL=0
MOVL C00550 V=800.0 PL=0
MOVL C00551 V=800.0 PL=0
MOVL C00552 V=800.0 PL=0
MOVL C00553 V=800.0 PL=0
MOVL C00554 V=800.0 PL=0
MOVL C00555 V=800.0 PL=0
MOVL C00556 V=800.0 PL=0
MOVL C00557 V=800.0 PL=0
MOVL C00558 V=800.0 PL=0
MOVL C00559 V=800.0 PL=0
MOVL C00560 V=800.0 PL=0
MOVL C00561 V=800.0 PL=0
MOVL C00562 V=800.0 PL=0
MOVL C00563 V=800.0 PL=0
MOVL C00564 V=800.0 PL=0
MOVL C00565 V=800.0 PL=0
MOVL C00566 V=800.0 PL=0
MOVL C00567 V=800.0 PL=0
MOVL C00568 V=800.0 PL=0
MOVL C00569 V=800.0 PL=0
MOVL C00570 V=800.0 PL=0
MOVL C00571 V=800.0 PL=0
MOVL C00572 V=800.0 PL=0
MOVL C00573 V=800.0 PL=0
MOVL C00574 V=800.0 PL=0
MOVL C00575 V=800.0 PL=0
MOVL C00576 V=800.0 PL=0
MOVL C00577 V=800.0 PL=0
MOVL C00578 V=800.0 PL=0
MOVL C00579 V=800.0 PL=0
MOVL C00580 V=800.0 PL=0
MOVL C00581 V=800.0 PL=0
MOVL C00582 V=800.0 PL=0
MOVL C00583 V=800.0 PL=0
MOVL C00584 V=800.0 PL=0
MOVL C00585 V=800.0 PL=0
MOVL C00586 V=800.0 PL=0
MOVL C00587 V=800.0 PL=0
MOVL C00588 V=800.0 PL=0
MOVL C00589 V=800.0 PL=0
MOVL C00590 V=800.0 PL=0
MOVL C00591 V=800.0 PL=0
MOVL C00592 V=800.0 PL=0
MOVL C00593 V=800.0 PL=0
MOVL C00594 V=800.0 PL=0
MOVL C00595 V=800.0 PL=0
MOVL C00596 V=800.0 PL=0
MOVL C00597 V=800.0 PL=0
MOVL C00598 V=800.0 PL=0
MOVL C00599 V=800.0 PL=0
MOVL C00600 V=800.0 PL=0
MOVL C00601 V=800.0 PL=0
MOVL C00602 V=800.0 PL=0
MOVL C00603 V=800.0 PL=0
MOVL C00604 V=800.0 PL=0
MOVL C00605 V=800.0 PL=0
MOVL C00606 V=800.0 PL=0
MOVL C00607 V=800.0 PL=0
MOVL C00608 V=800.0 PL=0
MOVL C00609 V=800.0 PL=0
MOVL C00610 V=800.0 PL=0
MOVL C00611 V=800.0 PL=0
MOVL C00612 V=800.0 PL=0
MOVL C00613 V=800.0 PL=0
MOVL C00614 V=800.0 PL=0
MOVL C00615 V=800.0 PL=0
MOVL C00616 V=800.0 PL=0
MOVL C00617 V=800.0 PL=0
MOVL C00618 V=800.0 PL=0
MOVL C00619 V=800.0 PL=0
MOVL C00620 V=800.0 PL=0
MOVL C00621 V=800.0 PL=0
MOVL C00622 V=800.0 PL=0
MOVL C00623 V=800.0 PL=0
MOVL C00624 V=800.0 PL=0
MOVL C00625 V=800.0 PL=0
MOVL C00626 V=800.0 PL=0
MOVL C00627 V=800.0 PL=0
MOVL C00628 V=800.0 PL=0
MOVL C00629 V=800.0 PL=0
MOVL C00630 V=800.0 PL=0
MOVL C00631 V=800.0 PL=0
MOVL C00632 V=800.0 PL=0
MOVL C00633 V=800.0 PL=0
MOVL C00634 V=800.0 PL=0
MOVL C00635 V=800.0 PL=0
MOVL C00636 V=800.0 PL=0
MOVL C00637 V=800.0 PL=0
MOVL C00638 V=800.0 PL=0
MOVL C00639 V=800.0 PL=0
MOVL C00640 V=800.0 PL=0
MOVL C00641 V=800.0 PL=0
MOVL C00642 V=800.0 PL=0
MOVL C00643 V=800.0 PL=0
MOVL C00644 V=800.0 PL=0
MOVL C00645 V=800.0 PL=0
MOVL C00646 V=800.0 PL=0
MOVL C00647 V=800.0 PL=0
MOVL C00648 V=800.0 PL=0
MOVL C00649 V=800.0 PL=0
MOVL C00650 V=800.0 PL=0
MOVL C00651 V=800.0 PL=0
MOVL C00652 V=800.0 PL=0
MOVL C00653 V=800.0 PL=0
MOVL C00654 V=800.0 PL=0
MOVL C00655 V=800.0 PL=0
MOVL C00656 V=800.0 PL=0
MOVL C00657 V=800.0 PL=0
MOVL C00658 V=800.0 PL=0
MOVL C00659 V=800.0 PL=0
MOVL C00660 V=800.0 PL=0
MOVL C00661 V=800.0 PL=0
MOVL C00662 V=800.0 PL=0
MOVL C00663 V=800.0 PL=0
MOVL C00664 V=800.0 PL=0
MOVL C00665 V=800.0 PL=0
MOVL C00666 V=800.0 PL=0
MOVL C00667 V=800.0 PL=0
MOVL C00668 V=800.0 PL=0
MOVL C00669 V=800.0 PL=0
MOVL C00670 V=800.0 PL=0
MOVL C00671 V=800.0 PL=0
MOVL C00672 V=800.0 PL=0
MOVL C00673 V=800.0 PL=0
MOVL C00674 V=800.0 PL=0
MOVL C00675 V=800.0 PL=0
MOVL C00676 V=800.0 PL=0
MOVL C00677 V=800.0 PL=0
MOVL C00678 V=800.0 PL=0
MOVL C00679 V=800.0 PL=0
MOVL C00680 V=800.0 PL=0
MOVL C00681 V=800.0 PL=0
MOVL C00682 V=800.0 PL=0
MOVL C00683 V=800.0 PL=0
MOVL C00684 V=800.0 PL=0
MOVL C00685 V=800.0 PL=0
MOVL C00686 V=800.0 PL=0
MOVL C00687 V=800.0 PL=0
MOVL C00688 V=800.0 PL=0
MOVL C00689 V=800.0 PL=0
MOVL C00690 V=800.0 PL=0
MOVL C00691 V=800.0 PL=0
MOVL C00692 V=800.0 PL=0
MOVL C00693 V=800.0 PL=0
MOVL C00694 V=800.0 PL=0
MOVL C00695 V=800.0 PL=0
MOVL C00696 V=800.0 PL=0
MOVL C00697 V=800.0 PL=0
MOVL C00698 V=800.0 PL=0
MOVL C00699 V=800.0 PL=0
MOVL C00700 V=800.0 PL=0
MOVL C00701 V=800.0 PL=0
MOVL C00702 V=800.0 PL=0
MOVL C00703 V=800.0 PL=0
MOVL C00704 V=800.0 PL=0
MOVL C00705 V=800.0 PL=0
MOVL C00706 V=800.0 PL=0
MOVL C00707 V=800.0 PL=0
MOVL C00708 V=800.0 PL=0
MOVL C00709 V=800.0 PL=0
MOVL C00710 V=800.0 PL=0
MOVL C00711 V=800.0 PL=0
MOVL C00712 V=800.0 PL=0
MOVL C00713 V=800.0 PL=0
MOVL C00714 V=800.0 PL=0
MOVL C00715 V=800.0 PL=0
MOVL C00716 V=800.0 PL=0
MOVL C00717 V=800.0 PL=0
MOVL C00718 V=800.0 PL=0
MOVL C00719 V=800.0 PL=0
MOVL C00720 V=800.0 PL=0
MOVL C00721 V=800.0 PL=0
MOVL C00722 V=800.0 PL=0
MOVL C00723 V=800.0 PL=0
MOVL C00724 V=800.0 PL=0
MOVL C00725 V=800.0 PL=0
MOVL C00726 V=800.0 PL=0
MOVL C00727 V=800.0 PL=0
MOVL C00728 V=800.0 PL=0
MOVL C00729 V=800.0 PL=0
MOVL C00730 V=800.0 PL=0
MOVL C00731 V=800.0 PL=0
MOVL C00732 V=800.0 PL=0
MOVL C00733 V=800.0 PL=0
MOVL C00734 V=800.0 PL=0
MOVL C00735 V=800.0 PL=0
MOVL C00736 V=800.0 PL=0
MOVL C00737 V=800.0 PL=0
MOVL C00738 V=800.0 PL=0
MOVL C00739 V=800.0 PL=0
MOVL C00740 V=800.0 PL=0
MOVL C00741 V=800.0 PL=0
MOVL C00742 V=800.0 PL=0
MOVL C00743 V=800.0 PL=0
MOVL C00744 V=800.0 PL=0
MOVL C00745 V=800.0 PL=0
MOVL C00746 V=800.0 PL=0
MOVL C00747 V=800.0 PL=0
MOVL C00748 V=800.0 PL=0
MOVL C00749 V=800.0 PL=0
MOVL C00750 V=800.0 PL=0
MOVL C00751 V=800.0 PL=0
MOVL C00752 V=800.0 PL=0
MOVL C00753 V=800.0 PL=0
MOVL C00754 V=800.0 PL=0
MOVL C00755 V=800.0 PL=0
MOVL C00756 V=800.0 PL=0
MOVL C00757 V=800.0 PL=0
MOVL C00758 V=800.0 PL=0
MOVL C00759 V=800.0 PL=0
MOVL C00760 V=800.0 PL=0
MOVL C00761 V=800.0 PL=0
MOVL C00762 V=800.0 PL=0
MOVL C00763 V=800.0 PL=0
MOVL C00764 V=800.0 PL=0
MOVL C00765 V=800.0 PL=0
MOVL C00766 V=800.0 PL=0
MOVL C00767 V=800.0 PL=0
MOVL C00768 V=800.0 PL=0
MOVL C00769 V=800.0 PL=0
MOVL C00770 V=800.0 PL=0
MOVL C00771 V=800.0 PL=0
MOVL C00772 V=800.0 PL=0
MOVL C00773 V=800.0 PL=0
MOVL C00774 V=800.0 PL=0
MOVL C00775 V=800.0 PL=0
MOVL C00776 V=800.0 PL=0
MOVL C00777 V=800.0 PL=0
MOVL C00778 V=800.0 PL=0
MOVL C00779 V=800.0 PL=0
MOVL C00780 V=800.0 PL=0
MOVL C00781 V=800.0 PL=0
MOVL C00782 V=800.0 PL=0
MOVL C00783 V=800.0 PL=0
MOVL C00784 V=800.0 PL=0
MOVL C00785 V=800.0 PL=0
MOVL C00786 V=800.0 PL=0
MOVL C00787 V=800.0 PL=0
MOVL C00788 V=800.0 PL=0
MOVL C00789 V=800.0 PL=0
MOVL C00790 V=800.0 PL=0
MOVL C00791 V=800.0 PL=0
MOVL C00792 V=800.0 PL=0
MOVL C00793 V=800.0 PL=0
MOVL C00794 V=800.0 PL=0
MOVL C00795 V=800.0 PL=0
MOVL C00796 V=800.0 PL=0
MOVL C00797 V=800.0 PL=0
MOVL C00798 V=800.0 PL=0
MOVL C00799 V=800.0 PL=0
MOVL C00800 V=800.0 PL=0
MOVL C00801 V=800.0 PL=0
MOVL C00802 V=800.0 PL=0
MOVL C00803 V=800.0 PL=0
MOVL C00804 V=800.0 PL=0
MOVL C00805 V=800.0 PL=0
MOVL C00806 V=800.0 PL=0
MOVL C00807 V=800.0 PL=0
MOVL C00808 V=800.0 PL=0
MOVL C00809 V=800.0 PL=0
MOVL C00810 V=800.0 PL=0
MOVL C00811 V=800.0 PL=0
MOVL C00812 V=800.0 PL=0
MOVL C00813 V=800.0 PL=0
MOVL C00814 V=800.0 PL=0
MOVL C00815 V=800.0 PL=0
MOVL C00816 V=800.0 PL=0
MOVL C00817 V=800.0 PL=0
MOVL C00818 V=800.0 PL=0
MOVL C00819 V=800.0 PL=0
MOVL C00820 V=800.0 PL=0
MOVL C00821 V=800.0 PL=0
MOVL C00822 V=800.0 PL=0
MOVL C00823 V=800.0 PL=0
MOVL C00824 V=800.0 PL=0
MOVL C00825 V=800.0 PL=0
MOVL C00826 V=800.0 PL=0
MOVL C00827 V=800.0 PL=0
MOVL C00828 V=800.0 PL=0
MOVL C00829 V=800.0 PL=0
MOVL C00830 V=800.0 PL=0
MOVL C00831 V=800.0 PL=0
MOVL C00832 V=800.0 PL=0
MOVL C00833 V=800.0 PL=0
MOVL C00834 V=800.0 PL=0
MOVL C00835 V=800.0 PL=0
MOVL C00836 V=800.0 PL=0
MOVL C00837 V=800.0 PL=0
MOVL C00838 V=800.0 PL=0
MOVL C00839 V=800.0 PL=0
MOVL C00840 V=800.0 PL=0
MOVL C00841 V=800.0 PL=0
MOVL C00842 V=800.0 PL=0
MOVL C00843 V=800.0 PL=0
MOVL C00844 V=800.0 PL=0
MOVL C00845 V=800.0 PL=0
MOVL C00846 V=800.0 PL=0
MOVL C00847 V=800.0 PL=0
MOVL C00848 V=800.0 PL=0
MOVL C00849 V=800.0 PL=0
MOVL C00850 V=800.0 PL=0
MOVL C00851 V=800.0 PL=0
MOVL C00852 V=800.0 PL=0
MOVL C00853 V=800.0 PL=0
MOVL C00854 V=800.0 PL=0
MOVL C00855 V=800.0 PL=0
MOVL C00856 V=800.0 PL=0
MOVL C00857 V=800.0 PL=0
MOVL C00858 V=800.0 PL=0
MOVL C00859 V=800.0 PL=0
MOVL C00860 V=800.0 PL=0
MOVL C00861 V=800.0 PL=0
MOVL C00862 V=800.0 PL=0
MOVL C00863 V=800.0 PL=0
MOVL C00864 V=800.0 PL=0
MOVL C00865 V=800.0 PL=0
MOVL C00866 V=800.0 PL=0
MOVL C00867 V=800.0 PL=0
MOVL C00868 V=800.0 PL=0
MOVL C00869 V=800.0 PL=0
MOVL C00870 V=800.0 PL=0
MOVL C00871 V=800.0 PL=0
MOVL C00872 V=800.0 PL=0
MOVL C00873 V=800.0 PL=0
MOVL C00874 V=800.0 PL=0
MOVL C00875 V=800.0 PL=0
MOVL C00876 V=800.0 PL=0
MOVL C00877 V=800.0 PL=0
MOVL C00878 V=800.0 PL=0
MOVL C00879 V=800.0 PL=0
MOVL C00880 V=800.0 PL=0
MOVL C00881 V=800.0 PL=0
MOVL C00882 V=800.0 PL=0
MOVL C00883 V=800.0 PL=0
MOVL C00884 V=800.0 PL=0
MOVL C00885 V=800.0 PL=0
MOVL C00886 V=800.0 PL=0
MOVL C00887 V=800.0 PL=0
MOVL C00888 V=800.0 PL=0
MOVL C00889 V=800.0 PL=0
MOVL C00890 V=800.0 PL=0
MOVL C00891 V=800.0 PL=0
MOVL C00892 V=800.0 PL=0
MOVL C00893 V=800.0 PL=0
MOVL C00894 V=800.0 PL=0
MOVL C00895 V=800.0 PL=0
MOVL C00896 V=800.0 PL=0
MOVL C00897 V=800.0 PL=0
MOVL C00898 V=800.0 PL=0
MOVL C00899 V=800.0 PL=0
MOVL C00900 V=800.0 PL=0
MOVL C00901 V=800.0 PL=0
MOVL C00902 V=800.0 PL=0
MOVL C00903 V=800.0 PL=0
MOVL C00904 V=800.0 PL=0
MOVL C00905 V=800.0 PL=0
MOVL C00906 V=800.0 PL=0
MOVL C00907 V=800.0 PL=0
MOVL C00908 V=800.0 PL=0
MOVL C00909 V=800.0 PL=0
MOVL C00910 V=800.0 PL=0
MOVL C00911 V=800.0 PL=0
MOVL C00912 V=800.0 PL=0
MOVL C00913 V=800.0 PL=0
MOVL C00914 V=800.0 PL=0
MOVL C00915 V=800.0 PL=0
MOVL C00916 V=800.0 PL=0
MOVL C00917 V=800.0 PL=0
MOVL C00918 V=800.0 PL=0
MOVL C00919 V=800.0 PL=0
MOVL C00920 V=800.0 PL=0
MOVL C00921 V=800.0 PL=0
MOVL C00922 V=800.0 PL=0
MOVL C00923 V=800.0 PL=0
MOVL C00924 V=800.0 PL=0
MOVL C00925 V=800.0 PL=0
MOVL C00926 V=800.0 PL=0
MOVL C00927 V=800.0 PL=0
MOVL C00928 V=800.0 PL=0
MOVL C00929 V=800.0 PL=0
MOVL C00930 V=800.0 PL=0
MOVL C00931 V=800.0 PL=0
MOVL C00932 V=800.0 PL=0
MOVL C00933 V=800.0 PL=0
MOVL C00934 V=800.0 PL=0
MOVL C00935 V=800.0 PL=0
MOVL C00936 V=800.0 PL=0
MOVL C00937 V=800.0 PL=0
MOVL C00938 V=800.0 PL=0
MOVL C00939 V=800.0 PL=0
MOVL C00940 V=800.0 PL=0
MOVL C00941 V=800.0 PL=0
MOVL C00942 V=800.0 PL=0
MOVL C00943 V=800.0 PL=0
MOVL C00944 V=800.0 PL=0
MOVL C00945 V=800.0 PL=0
MOVL C00946 V=800.0 PL=0
MOVL C00947 V=800.0 PL=0
MOVL C00948 V=800.0 PL=0
MOVL C00949 V=800.0 PL=0
MOVL C00950 V=800.0 PL=0
MOVL C00951 V=800.0 PL=0
MOVL C00952 V=800.0 PL=0
MOVL C00953 V=800.0 PL=0
MOVL C00954 V=800.0 PL=0
MOVL C00955 V=800.0 PL=0
MOVL C00956 V=800.0 PL=0
MOVL C00957 V=800.0 PL=0
MOVL C00958 V=800.0 PL=0
MOVL C00959 V=800.0 PL=0
MOVL C00960 V=800.0 PL=0
MOVL C00961 V=800.0 PL=0
MOVL C00962 V=800.0 PL=0
MOVL C00963 V=800.0 PL=0
MOVL C00964 V=800.0 PL=0
MOVL C00965 V=800.0 PL=0
MOVL C00966 V=800.0 PL=0
MOVL C00967 V=800.0 PL=0
MOVL C00968 V=800.0 PL=0
MOVL C00969 V=800.0 PL=0
MOVL C00970 V=800.0 PL=0
MOVL C00971 V=800.0 PL=0
MOVL C00972 V=800.0 PL=0
MOVL C00973 V=800.0 PL=0
MOVL C00974 V=800.0 PL=0
MOVL C00975 V=800.0 PL=0
MOVL C00976 V=800.0 PL=0
MOVL C00977 V=800.0 PL=0
MOVL C00978 V=800.0 PL=0
MOVL C00979 V=800.0 PL=0
MOVL C00980 V=800.0 PL=0
MOVL C00981 V=800.0 PL=0
MOVL C00982 V=800.0 PL=0
MOVL C00983 V=800.0 PL=0
MOVL C00984 V=800.0 PL=0
MOVL C00985 V=800.0 PL=0
MOVL C00986 V=800.0 PL=0
MOVL C00987 V=800.0 PL=0
MOVL C00988 V=800.0 PL=0
MOVL C00989 V=800.0 PL=0
MOVL C00990 V=800.0 PL=0
MOVL C00991 V=800.0 PL=0
MOVL C00992 V=800.0 PL=0
MOVL C00993 V=800.0 PL=0
MOVL C00994 V=800.0 PL=0
MOVL C00995 V=800.0 PL=0
MOVL C00996 V=800.0 PL=0
MOVL C00997 V=800.0 PL=0
MOVL C00998 V=800.0 PL=0
MOVL C00999 V=800.0 PL=0
MOVL C01000 V=800.0 PL=0
MOVL C01001 V=800.0 PL=0
MOVL C01002 V=800.0 PL=0
MOVL C01003 V=800.0 PL=0
MOVL C01004 V=800.0 PL=0
MOVL C01005 V=800.0 PL=0
MOVL C01006 V=800.0 PL=0
MOVL C01007 V=800.0 PL=0
MOVL C01008 V=800.0 PL=0
MOVL C01009 V=800.0 PL=0
MOVL C01010 V=800.0 PL=0
MOVL C01011 V=800.0 PL=0
MOVL C01012 V=800.0 PL=0
MOVL C01013 V=800.0 PL=0
MOVL C01014 V=800.0 PL=0
MOVL C01015 V=800.0 PL=0
MOVL C01016 V=800.0 PL=0
MOVL C01017 V=800.0 PL=0
MOVL C01018 V=800.0 PL=0
MOVL C01019 V=800.0 PL=0
MOVL C01020 V=800.0 PL=0
MOVL C01021 V=800.0 PL=0
MOVL C01022 V=800.0 PL=0
MOVL C01023 V=800.0 PL=0
MOVL C01024 V=800.0 PL=0
MOVL C01025 V=800.0 PL=0
MOVL C01026 V=800.0 PL=0
MOVL C01027 V=800.0 PL=0
MOVL C01028 V=800.0 PL=0
MOVL C01029 V=800.0 PL=0
MOVL C01030 V=800.0 PL=0
MOVL C01031 V=800.0 PL=0
MOVL C01032 V=800.0 PL=0
MOVL C01033 V=800.0 PL=0
MOVL C01034 V=800.0 PL=0
MOVL C01035 V=800.0 PL=0
MOVL C01036 V=800.0 PL=0
MOVL C01037 V=800.0 PL=0
MOVL C01038 V=800.0 PL=0
MOVL C01039 V=800.0 PL=0
MOVL C01040 V=800.0 PL=0
MOVL C01041 V=800.0 PL=0
MOVL C01042 V=800.0 PL=0
MOVL C01043 V=800.0 PL=0
MOVL C01044 V=800.0 PL=0
MOVL C01045 V=800.0 PL=0
MOVL C01046 V=800.0 PL=0
MOVL C01047 V=800.0 PL=0
MOVL C01048 V=800.0 PL=0
MOVL C01049 V=800.0 PL=0
MOVL C01050 V=800.0 PL=0
MOVL C01051 V=800.0 PL=0
MOVL C01052 V=800.0 PL=0
MOVL C01053 V=800.0 PL=0
MOVL C01054 V=800.0 PL=0
MOVL C01055 V=800.0 PL=0
MOVL C01056 V=800.0 PL=0
MOVL C01057 V=800.0 PL=0
MOVL C01058 V=800.0 PL=0
MOVL C01059 V=800.0 PL=0
MOVL C01060 V=800.0 PL=0
MOVL C01061 V=800.0 PL=0
MOVL C01062 V=800.0 PL=0
MOVL C01063 V=800.0 PL=0
MOVL C01064 V=800.0 PL=0
MOVL C01065 V=800.0 PL=0
MOVL C01066 V=800.0 PL=0
MOVL C01067 V=800.0 PL=0
MOVL C01068 V=800.0 PL=0
MOVL C01069 V=800.0 PL=0
MOVL C01070 V=800.0 PL=0
MOVL C01071 V=800.0 PL=0
MOVL C01072 V=800.0 PL=0
MOVL C01073 V=800.0 PL=0
MOVL C01074 V=800.0 PL=0
MOVL C01075 V=800.0 PL=0
MOVL C01076 V=800.0 PL=0
MOVL C01077 V=800.0 PL=0
MOVL C01078 V=800.0 PL=0
MOVL C01079 V=800.0 PL=0
MOVL C01080 V=800.0 PL=0
MOVL C01081 V=800.0 PL=0
MOVL C01082 V=800.0 PL=0
MOVL C01083 V=800.0 PL=0
MOVL C01084 V=800.0 PL=0
MOVL C01085 V=800.0 PL=0
MOVL C01086 V=800.0 PL=0
MOVL C01087 V=800.0 PL=0
MOVL C01088 V=800.0 PL=0
MOVL C01089 V=800.0 PL=0
MOVL C01090 V=800.0 PL=0
MOVL C01091 V=800.0 PL=0
MOVL C01092 V=800.0 PL=0
MOVL C01093 V=800.0 PL=0
MOVL C01094 V=800.0 PL=0
MOVL C01095 V=800.0 PL=0
MOVL C01096 V=800.0 PL=0
MOVL C01097 V=800.0 PL=0
MOVL C01098 V=800.0 PL=0
MOVL C01099 V=800.0 PL=0
MOVL C01100 V=800.0 PL=0
MOVL C01101 V=800.0 PL=0
MOVL C01102 V=800.0 PL=0
MOVL C01103 V=800.0 PL=0
MOVL C01104 V=800.0 PL=0
MOVL C01105 V=800.0 PL=0
MOVL C01106 V=800.0 PL=0
MOVL C01107 V=800.0 PL=0
MOVL C01108 V=800.0 PL=0
MOVL C01109 V=800.0 PL=0
MOVL C01110 V=800.0 PL=0
MOVL C01111 V=800.0 PL=0
MOVL C01112 V=800.0 PL=0
MOVL C01113 V=800.0 PL=0
MOVL C01114 V=800.0 PL=0
MOVL C01115 V=800.0 PL=0
MOVL C01116 V=800.0 PL=0
MOVL C01117 V=800.0 PL=0
MOVL C01118 V=800.0 PL=0
MOVL C01119 V=800.0 PL=0
MOVL C01120 V=800.0 PL=0
MOVL C01121 V=800.0 PL=0
MOVL C01122 V=800.0 PL=0
MOVL C01123 V=800.0 PL=0
MOVL C01124 V=800.0 PL=0
MOVL C01125 V=800.0 PL=0
MOVL C01126 V=800.0 PL=0
MOVL C01127 V=800.0 PL=0
MOVL C01128 V=800.0 PL=0
MOVL C01129 V=800.0 PL=0
MOVL C01130 V=800.0 PL=0
MOVL C01131 V=800.0 PL=0
MOVL C01132 V=800.0 PL=0
MOVL C01133 V=800.0 PL=0
MOVL C01134 V=800.0 PL=0
MOVL C01135 V=800.0 PL=0
MOVL C01136 V=800.0 PL=0
MOVL C01137 V=800.0 PL=0
MOVL C01138 V=800.0 PL=0
MOVL C01139 V=800.0 PL=0
MOVL C01140 V=800.0 PL=0
MOVL C01141 V=800.0 PL=0
MOVL C01142 V=800.0 PL=0
MOVL C01143 V=800.0 PL=0
MOVL C01144 V=800.0 PL=0
MOVL C01145 V=800.0 PL=0
MOVL C01146 V=800.0 PL=0
MOVL C01147 V=800.0 PL=0
MOVL C01148 V=800.0 PL=0
MOVL C01149 V=800.0 PL=0
MOVL C01150 V=800.0 PL=0
MOVL C01151 V=800.0 PL=0
MOVL C01152 V=800.0 PL=0
MOVL C01153 V=800.0 PL=0
MOVL C01154 V=800.0 PL=0
MOVL C01155 V=800.0 PL=0
MOVL C01156 V=800.0 PL=0
MOVL C01157 V=800.0 PL=0
MOVL C01158 V=800.0 PL=0
MOVL C01159 V=800.0 PL=0
MOVL C01160 V=800.0 PL=0
MOVL C01161 V=800.0 PL=0
MOVL C01162 V=800.0 PL=0
MOVL C01163 V=800.0 PL=0
MOVL C01164 V=800.0 PL=0
MOVL C01165 V=800.0 PL=0
MOVL C01166 V=800.0 PL=0
MOVL C01167 V=800.0 PL=0
MOVL C01168 V=800.0 PL=0
MOVL C01169 V=800.0 PL=0
MOVL C01170 V=800.0 PL=0
MOVL C01171 V=800.0 PL=0
MOVL C01172 V=800.0 PL=0
MOVL C01173 V=800.0 PL=0
MOVL C01174 V=800.0 PL=0
MOVL C01175 V=800.0 PL=0
MOVL C01176 V=800.0 PL=0
MOVL C01177 V=800.0 PL=0
MOVL C01178 V=800.0 PL=0
MOVL C01179 V=800.0 PL=0
MOVL C01180 V=800.0 PL=0
MOVL C01181 V=800.0 PL=0
MOVL C01182 V=800.0 PL=0
MOVL C01183 V=800.0 PL=0
MOVL C01184 V=800.0 PL=0
MOVL C01185 V=800.0 PL=0
MOVL C01186 V=800.0 PL=0
MOVL C01187 V=800.0 PL=0
MOVL C01188 V=800.0 PL=0
MOVL C01189 V=800.0 PL=0
MOVL C01190 V=800.0 PL=0
MOVL C01191 V=800.0 PL=0
MOVL C01192 V=800.0 PL=0
MOVL C01193 V=800.0 PL=0
MOVL C01194 V=800.0 PL=0
MOVL C01195 V=800.0 PL=0
MOVL C01196 V=800.0 PL=0
MOVL C01197 V=800.0 PL=0
MOVL C01198 V=800.0 PL=0
MOVL C01199 V=800.0 PL=0
MOVL C01200 V=800.0 PL=0
MOVL C01201 V=800.0 PL=0
MOVL C01202 V=800.0 PL=0
MOVL C01203 V=800.0 PL=0
MOVL C01204 V=800.0 PL=0
MOVL C01205 V=800.0 PL=0
MOVL C01206 V=800.0 PL=0
MOVL C01207 V=800.0 PL=0
MOVL C01208 V=800.0 PL=0
MOVL C01209 V=800.0 PL=0
MOVL C01210 V=800.0 PL=0
MOVL C01211 V=800.0 PL=0
MOVL C01212 V=800.0 PL=0
MOVL C01213 V=800.0 PL=0
MOVL C01214 V=800.0 PL=0
MOVL C01215 V=800.0 PL=0
MOVL C01216 V=800.0 PL=0
MOVL C01217 V=800.0 PL=0
MOVL C01218 V=800.0 PL=0
MOVL C01219 V=800.0 PL=0
MOVL C01220 V=800.0 PL=0
MOVL C01221 V=800.0 PL=0
MOVL C01222 V=800.0 PL=0
MOVL C01223 V=800.0 PL=0
MOVL C01224 V=800.0 PL=0
MOVL C01225 V=800.0 PL=0
MOVL C01226 V=800.0 PL=0
MOVL C01227 V=800.0 PL=0
MOVL C01228 V=800.0 PL=0
MOVL C01229 V=800.0 PL=0
MOVL C01230 V=800.0 PL=0
MOVL C01231 V=800.0 PL=0
MOVL C01232 V=800.0 PL=0
MOVL C01233 V=800.0 PL=0
MOVL C01234 V=800.0 PL=0
MOVL C01235 V=800.0 PL=0
MOVL C01236 V=800.0 PL=0
MOVL C01237 V=800.0 PL=0
MOVL C01238 V=800.0 PL=0
MOVL C01239 V=800.0 PL=0
MOVL C01240 V=800.0 PL=0
MOVL C01241 V=800.0 PL=0
MOVL C01242 V=800.0 PL=0
MOVL C01243 V=800.0 PL=0
MOVL C01244 V=800.0 PL=0
MOVL C01245 V=800.0 PL=0
MOVL C01246 V=800.0 PL=0
MOVL C01247 V=800.0 PL=0
MOVL C01248 V=800.0 PL=0
MOVL C01249 V=800.0 PL=0
MOVL C01250 V=800.0 PL=0
MOVL C01251 V=800.0 PL=0
MOVL C01252 V=800.0 PL=0
MOVL C01253 V=800.0 PL=0
MOVL C01254 V=800.0 PL=0
MOVL C01255 V=800.0 PL=0
MOVL C01256 V=800.0 PL=0
MOVL C01257 V=800.0 PL=0
MOVL C01258 V=800.0 PL=0
MOVL C01259 V=800.0 PL=0
MOVL C01260 V=800.0 PL=0
MOVL C01261 V=800.0 PL=0
MOVL C01262 V=800.0 PL=0
MOVL C01263 V=800.0 PL=0
MOVL C01264 V=800.0 PL=0
MOVL C01265 V=800.0 PL=0
MOVL C01266 V=800.0 PL=0
MOVL C01267 V=800.0 PL=0
MOVL C01268 V=800.0 PL=0
MOVL C01269 V=800.0 PL=0
MOVL C01270 V=800.0 PL=0
MOVL C01271 V=800.0 PL=0
MOVL C01272 V=800.0 PL=0
MOVL C01273 V=800.0 PL=0
MOVL C01274 V=800.0 PL=0
MOVL C01275 V=800.0 PL=0
MOVL C01276 V=800.0 PL=0
MOVL C01277 V=800.0 PL=0
MOVL C01278 V=800.0 PL=0
MOVL C01279 V=800.0 PL=0
MOVL C01280 V=800.0 PL=0
MOVL C01281 V=800.0 PL=0
MOVL C01282 V=800.0 PL=0
MOVL C01283 V=800.0 PL=0
MOVL C01284 V=800.0 PL=0
MOVL C01285 V=800.0 PL=0
MOVL C01286 V=800.0 PL=0
MOVL C01287 V=800.0 PL=0
MOVL C01288 V=800.0 PL=0
MOVL C01289 V=800.0 PL=0
MOVL C01290 V=800.0 PL=0
MOVL C01291 V=800.0 PL=0
MOVL C01292 V=800.0 PL=0
MOVL C01293 V=800.0 PL=0
MOVL C01294 V=800.0 PL=0
MOVL C01295 V=800.0 PL=0
MOVL C01296 V=800.0 PL=0
MOVL C01297 V=800.0 PL=0
MOVL C01298 V=800.0 PL=0
MOVL C01299 V=800.0 PL=0
MOVL C01300 V=800.0 PL=0
MOVL C01301 V=800.0 PL=0
MOVL C01302 V=800.0 PL=0
MOVL C01303 V=800.0 PL=0
MOVL C01304 V=800.0 PL=0
MOVL C01305 V=800.0 PL=0
MOVL C01306 V=800.0 PL=0
MOVL C01307 V=800.0 PL=0
MOVL C01308 V=800.0 PL=0
MOVL C01309 V=800.0 PL=0
MOVL C01310 V=800.0 PL=0
MOVL C01311 V=800.0 PL=0
MOVL C01312 V=800.0 PL=0
MOVL C01313 V=800.0 PL=0
MOVL C01314 V=800.0 PL=0
MOVL C01315 V=800.0 PL=0
MOVL C01316 V=800.0 PL=0
MOVL C01317 V=800.0 PL=0
MOVL C01318 V=800.0 PL=0
MOVL C01319 V=800.0 PL=0
MOVL C01320 V=800.0 PL=0
MOVL C01321 V=800.0 PL=0
MOVL C01322 V=800.0 PL=0
MOVL C01323 V=800.0 PL=0
MOVL C01324 V=800.0 PL=0
MOVL C01325 V=800.0 PL=0
MOVL C01326 V=800.0 PL=0
MOVL C01327 V=800.0 PL=0
MOVL C01328 V=800.0 PL=0
MOVL C01329 V=800.0 PL=0
MOVL C01330 V=800.0 PL=0
MOVL C01331 V=800.0 PL=0
MOVL C01332 V=800.0 PL=0
MOVL C01333 V=800.0 PL=0
MOVL C01334 V=800.0 PL=0
MOVL C01335 V=800.0 PL=0
MOVL C01336 V=800.0 PL=0
MOVL C01337 V=800.0 PL=0
MOVL C01338 V=800.0 PL=0
MOVL C01339 V=800.0 PL=0
MOVL C01340 V=800.0 PL=0
MOVL C01341 V=800.0 PL=0
MOVL C01342 V=800.0 PL=0
MOVL C01343 V=800.0 PL=0
MOVL C01344 V=800.0 PL=0
MOVL C01345 V=800.0 PL=0
MOVL C01346 V=800.0 PL=0
MOVL C01347 V=800.0 PL=0
MOVL C01348 V=800.0 PL=0
MOVL C01349 V=800.0 PL=0
MOVL C01350 V=800.0 PL=0
MOVL C01351 V=800.0 PL=0
MOVL C01352 V=800.0 PL=0
MOVL C01353 V=800.0 PL=0
MOVL C01354 V=800.0 PL=0
MOVL C01355 V=800.0 PL=0
MOVL C01356 V=800.0 PL=0
MOVL C01357 V=800.0 PL=0
MOVL C01358 V=800.0 PL=0
MOVL C01359 V=800.0 PL=0
MOVL C01360 V=800.0 PL=0
MOVL C01361 V=800.0 PL=0
MOVL C01362 V=800.0 PL=0
MOVL C01363 V=800.0 PL=0
MOVL C01364 V=800.0 PL=0
MOVL C01365 V=800.0 PL=0
MOVL C01366 V=800.0 PL=0
MOVL C01367 V=800.0 PL=0
MOVL C01368 V=800.0 PL=0
MOVL C01369 V=800.0 PL=0
MOVL C01370 V=800.0 PL=0
MOVL C01371 V=800.0 PL=0
MOVL C01372 V=800.0 PL=0
MOVL C01373 V=800.0 PL=0
MOVL C01374 V=800.0 PL=0
MOVL C01375 V=800.0 PL=0
MOVL C01376 V=800.0 PL=0
MOVL C01377 V=800.0 PL=0
MOVL C01378 V=800.0 PL=0
MOVL C01379 V=800.0 PL=0
MOVL C01380 V=800.0 PL=0
MOVL C01381 V=800.0 PL=0
MOVL C01382 V=800.0 PL=0
MOVL C01383 V=800.0 PL=0
MOVL C01384 V=800.0 PL=0
MOVL C01385 V=800.0 PL=0
MOVL C01386 V=800.0 PL=0
MOVL C01387 V=800.0 PL=0
MOVL C01388 V=800.0 PL=0
MOVL C01389 V=800.0 PL=0
MOVL C01390 V=800.0 PL=0
MOVL C01391 V=800.0 PL=0
MOVL C01392 V=800.0 PL=0
MOVL C01393 V=800.0 PL=0
MOVL C01394 V=800.0 PL=0
MOVL C01395 V=800.0 PL=0
MOVL C01396 V=800.0 PL=0
MOVL C01397 V=800.0 PL=0
MOVL C01398 V=800.0 PL=0
MOVL C01399 V=800.0 PL=0
MOVL C01400 V=800.0 PL=0
MOVL C01401 V=800.0 PL=0
MOVL C01402 V=800.0 PL=0
MOVL C01403 V=800.0 PL=0
MOVL C01404 V=800.0 PL=0
MOVL C01405 V=800.0 PL=0
MOVL C01406 V=800.0 PL=0
MOVL C01407 V=800.0 PL=0
MOVL C01408 V=800.0 PL=0
MOVL C01409 V=800.0 PL=0
MOVL C01410 V=800.0 PL=0
MOVL C01411 V=800.0 PL=0
MOVL C01412 V=800.0 PL=0
MOVL C01413 V=800.0 PL=0
MOVL C01414 V=800.0 PL=0
MOVL C01415 V=800.0 PL=0
MOVL C01416 V=800.0 PL=0
MOVL C01417 V=800.0 PL=0
MOVL C01418 V=800.0 PL=0
MOVL C01419 V=800.0 PL=0
MOVL C01420 V=800.0 PL=0
MOVL C01421 V=800.0 PL=0
MOVL C01422 V=800.0 PL=0
MOVL C01423 V=800.0 PL=0
MOVL C01424 V=800.0 PL=0
MOVL C01425 V=800.0 PL=0
MOVL C01426 V=800.0 PL=0
MOVL C01427 V=800.0 PL=0
MOVL C01428 V=800.0 PL=0
MOVL C01429 V=800.0 PL=0
MOVL C01430 V=800.0 PL=0
MOVL C01431 V=800.0 PL=0
MOVL C01432 V=800.0 PL=0
MOVL C01433 V=800.0 PL=0
MOVL C01434 V=800.0 PL=0
MOVL C01435 V=800.0 PL=0
MOVL C01436 V=800.0 PL=0
MOVL C01437 V=800.0 PL=0
MOVL C01438 V=800.0 PL=0
MOVL C01439 V=800.0 PL=0
MOVL C01440 V=800.0 PL=0
MOVL C01441 V=800.0 PL=0
MOVL C01442 V=800.0 PL=0
MOVL C01443 V=800.0 PL=0
MOVL C01444 V=800.0 PL=0
MOVL C01445 V=800.0 PL=0
MOVL C01446 V=800.0 PL=0
MOVL C01447 V=800.0 PL=0
MOVL C01448 V=800.0 PL=0
MOVL C01449 V=800.0 PL=0
MOVL C01450 V=800.0 PL=0
MOVL C01451 V=800.0 PL=0
MOVL C01452 V=800.0 PL=0
MOVL C01453 V=800.0 PL=0
MOVL C01454 V=800.0 PL=0
MOVL C01455 V=800.0 PL=0
MOVL C01456 V=800.0 PL=0
MOVL C01457 V=800.0 PL=0
MOVL C01458 V=800.0 PL=0
MOVL C01459 V=800.0 PL=0
MOVL C01460 V=800.0 PL=0
MOVL C01461 V=800.0 PL=0
MOVL C01462 V=800.0 PL=0
MOVL C01463 V=800.0 PL=0
MOVL C01464 V=800.0 PL=0
MOVL C01465 V=800.0 PL=0
MOVL C01466 V=800.0 PL=0
MOVL C01467 V=800.0 PL=0
MOVL C01468 V=800.0 PL=0
MOVL C01469 V=800.0 PL=0
MOVL C01470 V=800.0 PL=0
MOVL C01471 V=800.0 PL=0
MOVL C01472 V=800.0 PL=0
MOVL C01473 V=800.0 PL=0
MOVL C01474 V=800.0 PL=0
MOVL C01475 V=800.0 PL=0
MOVL C01476 V=800.0 PL=0
MOVL C01477 V=800.0 PL=0
MOVL C01478 V=800.0 PL=0
MOVL C01479 V=800.0 PL=0
MOVL C01480 V=800.0 PL=0
MOVL C01481 V=800.0 PL=0
MOVL C01482 V=800.0 PL=0
MOVL C01483 V=800.0 PL=0
MOVL C01484 V=800.0 PL=0
MOVL C01485 V=800.0 PL=0
MOVL C01486 V=800.0 PL=0
MOVL C01487 V=800.0 PL=0
MOVL C01488 V=800.0 PL=0
MOVL C01489 V=800.0 PL=0
MOVL C01490 V=800.0 PL=0
MOVL C01491 V=800.0 PL=0
MOVL C01492 V=800.0 PL=0
MOVL C01493 V=800.0 PL=0
MOVL C01494 V=800.0 PL=0
MOVL C01495 V=800.0 PL=0
MOVL C01496 V=800.0 PL=0
MOVL C01497 V=800.0 PL=0
MOVL C01498 V=800.0 PL=0
MOVL C01499 V=800.0 PL=0
MOVL C01500 V=800.0 PL=0
MOVL C01501 V=800.0 PL=0
MOVL C01502 V=800.0 PL=0
MOVL C01503 V=800.0 PL=0
MOVL C01504 V=800.0 PL=0
MOVL C01505 V=800.0 PL=0
MOVL C01506 V=800.0 PL=0
MOVL C01507 V=800.0 PL=0
MOVL C01508 V=800.0 PL=0
MOVL C01509 V=800.0 PL=0
MOVL C01510 V=800.0 PL=0
MOVL C01511 V=800.0 PL=0
MOVL C01512 V=800.0 PL=0
MOVL C01513 V=800.0 PL=0
MOVL C01514 V=800.0 PL=0
MOVL C01515 V=800.0 PL=0
MOVL C01516 V=800.0 PL=0
MOVL C01517 V=800.0 PL=0
MOVL C01518 V=800.0 PL=0
MOVL C01519 V=800.0 PL=0
MOVL C01520 V=800.0 PL=0
MOVL C01521 V=800.0 PL=0
MOVL C01522 V=800.0 PL=0
MOVL C01523 V=800.0 PL=0
MOVL C01524 V=800.0 PL=0
MOVL C01525 V=800.0 PL=0
MOVL C01526 V=800.0 PL=0
MOVL C01527 V=800.0 PL=0
MOVL C01528 V=800.0 PL=0
MOVL C01529 V=800.0 PL=0
MOVL C01530 V=800.0 PL=0
MOVL C01531 V=800.0 PL=0
MOVL C01532 V=800.0 PL=0
MOVL C01533 V=800.0 PL=0
MOVL C01534 V=800.0 PL=0
MOVL C01535 V=800.0 PL=0
MOVL C01536 V=800.0 PL=0
MOVL C01537 V=800.0 PL=0
MOVL C01538 V=800.0 PL=0
MOVL C01539 V=800.0 PL=0
MOVL C01540 V=800.0 PL=0
MOVL C01541 V=800.0 PL=0
MOVL C01542 V=800.0 PL=0
MOVL C01543 V=800.0 PL=0
MOVL C01544 V=800.0 PL=0
MOVL C01545 V=800.0 PL=0
MOVL C01546 V=800.0 PL=0
MOVL C01547 V=800.0 PL=0
MOVL C01548 V=800.0 PL=0
MOVL C01549 V=800.0 PL=0
MOVL C01550 V=800.0 PL=0
MOVL C01551 V=800.0 PL=0
MOVL C01552 V=800.0 PL=0
MOVL C01553 V=800.0 PL=0
MOVL C01554 V=800.0 PL=0
MOVL C01555 V=800.0 PL=0
MOVL C01556 V=800.0 PL=0
MOVL C01557 V=800.0 PL=0
MOVL C01558 V=800.0 PL=0
MOVL C01559 V=800.0 PL=0
MOVL C01560 V=800.0 PL=0
MOVL C01561 V=800.0 PL=0
MOVL C01562 V=800.0 PL=0
MOVL C01563 V=800.0 PL=0
MOVL C01564 V=800.0 PL=0
MOVL C01565 V=800.0 PL=0
MOVL C01566 V=800.0 PL=0
MOVL C01567 V=800.0 PL=0
MOVL C01568 V=800.0 PL=0
MOVL C01569 V=800.0 PL=0
MOVL C01570 V=800.0 PL=0
MOVL C01571 V=800.0 PL=0
MOVL C01572 V=800.0 PL=0
MOVL C01573 V=800.0 PL=0
MOVL C01574 V=800.0 PL=0
MOVL C01575 V=800.0 PL=0
MOVL C01576 V=800.0 PL=0
MOVL C01577 V=800.0 PL=0
MOVL C01578 V=800.0 PL=0
MOVL C01579 V=800.0 PL=0
MOVL C01580 V=800.0 PL=0
MOVL C01581 V=800.0 PL=0
MOVL C01582 V=800.0 PL=0
MOVL C01583 V=800.0 PL=0
MOVL C01584 V=800.0 PL=0
MOVL C01585 V=800.0 PL=0
MOVL C01586 V=800.0 PL=0
MOVL C01587 V=800.0 PL=0
MOVL C01588 V=800.0 PL=0
MOVL C01589 V=800.0 PL=0
MOVL C01590 V=800.0 PL=0
MOVL C01591 V=800.0 PL=0
MOVL C01592 V=800.0 PL=0
MOVL C01593 V=800.0 PL=0
MOVL C01594 V=800.0 PL=0
MOVL C01595 V=800.0 PL=0
MOVL C01596 V=800.0 PL=0
MOVL C01597 V=800.0 PL=0
MOVL C01598 V=800.0 PL=0
MOVL C01599 V=800.0 PL=0
MOVL C01600 V=800.0 PL=0
MOVL C01601 V=800.0 PL=0
MOVL C01602 V=800.0 PL=0
MOVL C01603 V=800.0 PL=0
MOVL C01604 V=800.0 PL=0
MOVL C01605 V=800.0 PL=0
MOVL C01606 V=800.0 PL=0
MOVL C01607 V=800.0 PL=0
MOVL C01608 V=800.0 PL=0
MOVL C01609 V=800.0 PL=0
MOVL C01610 V=800.0 PL=0
MOVL C01611 V=800.0 PL=0
MOVL C01612 V=800.0 PL=0
MOVL C01613 V=800.0 PL=0
MOVL C01614 V=800.0 PL=0
MOVL C01615 V=800.0 PL=0
MOVL C01616 V=800.0 PL=0
MOVL C01617 V=800.0 PL=0
MOVL C01618 V=800.0 PL=0
MOVL C01619 V=800.0 PL=0
MOVL C01620 V=800.0 PL=0
MOVL C01621 V=800.0 PL=0
MOVL C01622 V=800.0 PL=0
MOVL C01623 V=800.0 PL=0
MOVL C01624 V=800.0 PL=0
MOVL C01625 V=800.0 PL=0
MOVL C01626 V=800.0 PL=0
MOVL C01627 V=800.0 PL=0
MOVL C01628 V=800.0 PL=0
MOVL C01629 V=800.0 PL=0
MOVL C01630 V=800.0 PL=0
MOVL C01631 V=800.0 PL=0
MOVL C01632 V=800.0 PL=0
MOVL C01633 V=800.0 PL=0
MOVL C01634 V=800.0 PL=0
MOVL C01635 V=800.0 PL=0
MOVL C01636 V=800.0 PL=0
MOVL C01637 V=800.0 PL=0
MOVL C01638 V=800.0 PL=0
MOVL C01639 V=800.0 PL=0
MOVL C01640 V=800.0 PL=0
MOVL C01641 V=800.0 PL=0
MOVL C01642 V=800.0 PL=0
MOVL C01643 V=800.0 PL=0
